LIN {X -0.179,Y -370.669,Z 1236.439,A 0.000,B 0.000,C 90.000,E1 79.106} C_DIS
LIN {X 0.099,Y -361.272,Z 1236.430,A 0.000,B 0.000,C 90.000,E1 77.297} C_DIS
LIN {X 0.011,Y -351.626,Z 1236.420,A 0.000,B 0.000,C 90.000,E1 75.519} C_DIS
LIN {X 0.097,Y -340.229,Z 1236.408,A 0.000,B 0.000,C 90.000,E1 73.378} C_DIS
LIN {X 0.001,Y -327.542,Z 1236.394,A 0.000,B 0.000,C 90.000,E1 70.913} C_DIS
LIN {X 0.007,Y -310.788,Z 1236.375,A 0.000,B 0.000,C 90.000,E1 67.411} C_DIS
LIN {X -0.044,Y -295.583,Z 1236.354,A 0.000,B 0.000,C 90.000,E1 63.819} C_DIS
LIN {X -0.046,Y -282.943,Z 1236.336,A 0.000,B 0.000,C 90.000,E1 60.461} C_DIS
LIN {X -0.122,Y -271.304,Z 1236.317,A 0.000,B 0.000,C 90.000,E1 57.041} C_DIS
LIN {X 0.053,Y -260.652,Z 1236.297,A 0.000,B 0.000,C 90.000,E1 53.497} C_DIS
LIN {X 0.109,Y -250.938,Z 1236.277,A 0.000,B 0.000,C 90.000,E1 49.908} C_DIS
LIN {X -0.029,Y -241.950,Z 1236.257,A 0.000,B 0.000,C 90.000,E1 46.296} C_DIS
LIN {X -0.042,Y -235.054,Z 1236.241,A 0.000,B 0.000,C 90.000,E1 43.338} C_DIS
LIN {X -0.040,Y -228.349,Z 1236.224,A 0.000,B 0.000,C 90.000,E1 40.334} C_DIS
LIN {X 0.029,Y -220.435,Z 1236.203,A 0.000,B 0.000,C 90.000,E1 36.503} C_DIS
LIN {X 0.039,Y -213.341,Z 1236.181,A 0.000,B 0.000,C 90.000,E1 32.625} C_DIS
LIN {X 0.035,Y -207.183,Z 1236.159,A 0.000,B 0.000,C 90.000,E1 28.693} C_DIS
LIN {X -0.003,Y -201.815,Z 1236.137,A 0.000,B 0.000,C 90.000,E1 24.719} C_DIS
LIN {X 0.088,Y -197.451,Z 1236.115,A 0.000,B 0.000,C 90.000,E1 20.663} C_DIS
LIN {X 0.056,Y -193.292,Z 1236.088,A 0.000,B 0.000,C 90.000,E1 15.788} C_DIS
LIN {X -0.068,Y -190.051,Z 1236.056,A 0.000,B 0.000,C 90.000,E1 10.074} C_DIS
LIN {X -0.056,Y -190.199,Z 1235.974,A 0.000,B 0.000,C 90.000,E1 355.412} C_DIS
LIN {X -0.017,Y -193.411,Z 1235.942,A 0.000,B 0.000,C 90.000,E1 349.634} C_DIS
LIN {X -0.111,Y -197.411,Z 1235.915,A 0.000,B 0.000,C 90.000,E1 344.755} C_DIS
LIN {X -0.029,Y -201.638,Z 1235.893,A 0.000,B 0.000,C 90.000,E1 340.678} C_DIS
LIN {X -0.040,Y -206.594,Z 1235.870,A 0.000,B 0.000,C 90.000,E1 336.666} C_DIS
LIN {X 0.069,Y -212.254,Z 1235.848,A 0.000,B 0.000,C 90.000,E1 332.666} C_DIS
LIN {X 0.023,Y -217.130,Z 1235.831,A 0.000,B 0.000,C 90.000,E1 329.537} C_DIS
LIN {X -0.042,Y -223.851,Z 1235.809,A 0.000,B 0.000,C 90.000,E1 325.674} C_DIS
LIN {X 0.063,Y -231.206,Z 1235.788,A 0.000,B 0.000,C 90.000,E1 321.823} C_DIS
LIN {X -0.030,Y -239.421,Z 1235.767,A 0.000,B 0.000,C 90.000,E1 318.081} C_DIS
LIN {X -0.074,Y -247.766,Z 1235.749,A 0.000,B 0.000,C 90.000,E1 314.757} C_DIS
LIN {X -0.018,Y -257.363,Z 1235.730,A 0.000,B 0.000,C 90.000,E1 311.472} C_DIS
LIN {X 0.156,Y -263.424,Z 1235.720,A 0.000,B 0.000,C 90.000,E1 309.644} C_DIS
LIN {X -0.140,Y -273.079,Z 1235.707,A 0.000,B 0.000,C 90.000,E1 307.237} C_DIS
LIN {X -0.057,Y -285.485,Z 1235.691,A 0.000,B 0.000,C 90.000,E1 304.452} C_DIS
LIN {X -0.050,Y -295.886,Z 1235.680,A 0.000,B 0.000,C 90.000,E1 302.418} C_DIS
LIN {X -0.011,Y -305.286,Z 1235.671,A 0.000,B 0.000,C 90.000,E1 300.747} C_DIS
LIN {X 0.082,Y -311.517,Z 1235.665,A 0.000,B 0.000,C 90.000,E1 299.745} C_DIS
LIN {X -0.191,Y -318.308,Z 1235.660,A 0.000,B 0.000,C 90.000,E1 298.821} C_DIS
LIN {X -0.131,Y -340.816,Z 1235.644,A 0.000,B 0.000,C 90.000,E1 295.976} C_DIS
LIN {X 0.057,Y -356.578,Z 1235.634,A 0.000,B 0.000,C 90.000,E1 294.131} C_DIS
LIN {X -0.042,Y -374.823,Z 1235.623,A 0.000,B 0.000,C 90.000,E1 292.153} C_DIS
LIN {X -0.141,Y -390.434,Z 1235.614,A 0.000,B 0.000,C 90.000,E1 290.482} C_DIS
LIN {X 0.066,Y -408.526,Z 1235.603,A 0.000,B 0.000,C 90.000,E1 288.544} C_DIS
LIN {X 0.208,Y -418.729,Z 1235.597,A 0.000,B 0.000,C 90.000,E1 287.457} C_DIS
LIN {X 0.098,Y -426.028,Z 1235.593,A 0.000,B 0.000,C 90.000,E1 286.677} C_DIS
LIN {X -0.103,Y -432.907,Z 1235.588,A 0.000,B 0.000,C 90.000,E1 285.898} C_DIS
LIN {X 0.145,Y -439.240,Z 1235.584,A 0.000,B 0.000,C 90.000,E1 285.064} C_DIS
LIN {X -0.092,Y -445.008,Z 1235.579,A 0.000,B 0.000,C 90.000,E1 284.300} C_DIS
LIN {X 0.164,Y -450.121,Z 1235.575,A 0.000,B 0.000,C 90.000,E1 283.480} C_DIS
LIN {X 0.027,Y -454.497,Z 1235.571,A 0.000,B 0.000,C 90.000,E1 282.715} C_DIS
LIN {X -0.069,Y -458.168,Z 1235.566,A 0.000,B 0.000,C 90.000,E1 281.951} C_DIS
LIN {X -0.139,Y -461.249,Z 1235.562,A 0.000,B 0.000,C 90.000,E1 281.186} C_DIS
LIN {X -0.027,Y -463.002,Z 1235.559,A 0.000,B 0.000,C 90.000,E1 280.658} C_DIS
LIN {X 0.014,Y -464.458,Z 1235.556,A 0.000,B 0.000,C 90.000,E1 280.141} C_DIS
LIN {X 0.148,Y -465.715,Z 1235.553,A 0.000,B 0.000,C 90.000,E1 279.613} C_DIS
LIN {X -0.247,Y -466.684,Z 1235.551,A 0.000,B 0.000,C 90.000,E1 279.151} C_DIS
LIN {X -0.102,Y -467.333,Z 1235.548,A 0.000,B 0.000,C 90.000,E1 278.624} C_DIS
LIN {X -0.024,Y -467.672,Z 1235.545,A 0.000,B 0.000,C 90.000,E1 278.106} C_DIS
LIN {X 0.062,Y -467.688,Z 1235.542,A 0.000,B 0.000,C 90.000,E1 277.587} C_DIS
LIN {X 0.152,Y -467.320,Z 1235.539,A 0.000,B 0.000,C 90.000,E1 277.068} C_DIS
LIN {X -0.222,Y -466.486,Z 1235.536,A 0.000,B 0.000,C 90.000,E1 276.606} C_DIS
LIN {X -0.133,Y -465.262,Z 1235.534,A 0.000,B 0.000,C 90.000,E1 276.087} C_DIS
LIN {X -0.051,Y -463.627,Z 1235.531,A 0.000,B 0.000,C 90.000,E1 275.568} C_DIS
LIN {X 0.023,Y -461.532,Z 1235.528,A 0.000,B 0.000,C 90.000,E1 275.049} C_DIS
LIN {X 0.086,Y -458.948,Z 1235.525,A 0.000,B 0.000,C 90.000,E1 274.531} C_DIS
LIN {X -0.139,Y -457.507,Z 1235.524,A 0.000,B 0.000,C 90.000,E1 274.302} C_DIS
LIN {X -0.105,Y -453.967,Z 1235.521,A 0.000,B 0.000,C 90.000,E1 273.784} C_DIS
LIN {X 0.119,Y -451.884,Z 1235.520,A 0.000,B 0.000,C 90.000,E1 273.498} C_DIS
LIN {X 0.119,Y -446.831,Z 1235.517,A 0.000,B 0.000,C 90.000,E1 272.980} C_DIS
LIN {X -0.189,Y -440.738,Z 1235.514,A 0.000,B 0.000,C 90.000,E1 272.522} C_DIS
LIN {X 0.061,Y -434.052,Z 1235.511,A 0.000,B 0.000,C 90.000,E1 272.064} C_DIS
LIN {X 0.003,Y -427.110,Z 1235.510,A 0.000,B 0.000,C 90.000,E1 271.718} C_DIS
LIN {X -0.030,Y -420.025,Z 1235.508,A 0.000,B 0.000,C 90.000,E1 271.432} C_DIS
LIN {X -0.120,Y -412.965,Z 1235.507,A 0.000,B 0.000,C 90.000,E1 271.203} C_DIS
LIN {X 0.061,Y -405.743,Z 1235.505,A 0.000,B 0.000,C 90.000,E1 270.974} C_DIS
LIN {X -0.013,Y -395.190,Z 1235.504,A 0.000,B 0.000,C 90.000,E1 270.745} C_DIS
LIN {X -0.148,Y -387.567,Z 1235.503,A 0.000,B 0.000,C 90.000,E1 270.630} C_DIS
LIN {X -0.120,Y -378.532,Z 1235.503,A 0.000,B 0.000,C 90.000,E1 270.516} C_DIS
LIN {X 0.140,Y -365.055,Z 1235.502,A 0.000,B 0.000,C 90.000,E1 270.401} C_DIS
LIN {X 0.082,Y -359.253,Z 1235.502,A 0.000,B 0.000,C 90.000,E1 270.401} C_DIS
LIN {X 0.013,Y -181.576,Z 1235.502,A 0.000,B 0.000,C 90.000,E1 270.401} C_DIS
LIN {X -0.055,Y -180.860,Z 1235.472,A 0.000,B 0.000,C 90.000,E1 265.008} C_DIS
LIN {X -0.001,Y -178.972,Z 1235.444,A 0.000,B 0.000,C 90.000,E1 259.926} C_DIS
LIN {X 0.008,Y -177.932,Z 1235.435,A 0.000,B 0.000,C 90.000,E1 258.229} C_DIS
LIN {X 0.024,Y -175.570,Z 1235.411,A 0.000,B 0.000,C 90.000,E1 253.976} C_DIS
LIN {X 0.030,Y -172.299,Z 1235.387,A 0.000,B 0.000,C 90.000,E1 249.699} C_DIS
LIN {X 0.008,Y -171.777,Z 1235.382,A 0.000,B 0.000,C 90.000,E1 248.847} C_DIS
LIN {X -0.020,Y -168.707,Z 1235.363,A 0.000,B 0.000,C 90.000,E1 245.409} C_DIS
LIN {X 0.019,Y -166.770,Z 1235.349,A 0.000,B 0.000,C 90.000,E1 242.794} C_DIS
LIN {X -0.061,Y -162.751,Z 1235.325,A 0.000,B 0.000,C 90.000,E1 238.456} C_DIS
LIN {X -0.085,Y -161.441,Z 1235.315,A 0.000,B 0.000,C 90.000,E1 236.707} C_DIS
LIN {X -0.042,Y -157.434,Z 1235.290,A 0.000,B 0.000,C 90.000,E1 232.271} C_DIS
LIN {X -0.009,Y -155.440,Z 1235.276,A 0.000,B 0.000,C 90.000,E1 229.585} C_DIS
LIN {X 0.040,Y -151.761,Z 1235.250,A 0.000,B 0.000,C 90.000,E1 225.081} C_DIS
LIN {X 0.052,Y -149.962,Z 1235.235,A 0.000,B 0.000,C 90.000,E1 222.366} C_DIS
LIN {X 0.079,Y -146.802,Z 1235.210,A 0.000,B 0.000,C 90.000,E1 217.810} C_DIS
LIN {X -0.021,Y -145.379,Z 1235.195,A 0.000,B 0.000,C 90.000,E1 215.105} C_DIS
LIN {X -0.029,Y -142.440,Z 1235.164,A 0.000,B 0.000,C 90.000,E1 209.589} C_DIS
LIN {X 0.018,Y -141.431,Z 1235.149,A 0.000,B 0.000,C 90.000,E1 206.796} C_DIS
LIN {X -0.001,Y -139.365,Z 1235.113,A 0.000,B 0.000,C 90.000,E1 200.301} C_DIS
LIN {X -0.015,Y -138.810,Z 1235.097,A 0.000,B 0.000,C 90.000,E1 197.511} C_DIS
LIN {X 0.037,Y -138.351,Z 1235.056,A 0.000,B 0.000,C 90.000,E1 190.018} C_DIS
LIN {X 0.012,Y -139.540,Z 1235.004,A 0.000,B 0.000,C 90.000,E1 180.688} C_DIS
LIN {X -0.035,Y -141.237,Z 1234.973,A 0.000,B 0.000,C 90.000,E1 175.122} C_DIS
LIN {X 0.065,Y -142.607,Z 1234.957,A 0.000,B 0.000,C 90.000,E1 172.299} C_DIS
LIN {X 0.018,Y -144.918,Z 1234.932,A 0.000,B 0.000,C 90.000,E1 167.701} C_DIS
LIN {X 0.010,Y -147.547,Z 1234.911,A 0.000,B 0.000,C 90.000,E1 164.031} C_DIS
LIN {X 0.042,Y -150.149,Z 1234.891,A 0.000,B 0.000,C 90.000,E1 160.369} C_DIS
LIN {X 0.052,Y -153.518,Z 1234.871,A 0.000,B 0.000,C 90.000,E1 156.741} C_DIS
LIN {X -0.027,Y -157.883,Z 1234.846,A 0.000,B 0.000,C 90.000,E1 152.281} C_DIS
LIN {X -0.073,Y -162.170,Z 1234.826,A 0.000,B 0.000,C 90.000,E1 148.742} C_DIS
LIN {X 0.042,Y -166.379,Z 1234.807,A 0.000,B 0.000,C 90.000,E1 145.182} C_DIS
LIN {X 0.044,Y -171.395,Z 1234.787,A 0.000,B 0.000,C 90.000,E1 141.698} C_DIS
LIN {X 0.084,Y -176.308,Z 1234.768,A 0.000,B 0.000,C 90.000,E1 138.243} C_DIS
LIN {X -0.047,Y -180.595,Z 1234.754,A 0.000,B 0.000,C 90.000,E1 135.729} C_DIS
LIN {X -0.070,Y -185.996,Z 1234.735,A 0.000,B 0.000,C 90.000,E1 132.366} C_DIS
LIN {X -0.015,Y -190.631,Z 1234.721,A 0.000,B 0.000,C 90.000,E1 129.850} C_DIS
LIN {X -0.108,Y -196.381,Z 1234.703,A 0.000,B 0.000,C 90.000,E1 126.583} C_DIS
LIN {X -0.039,Y -200.820,Z 1234.691,A 0.000,B 0.000,C 90.000,E1 124.326} C_DIS
LIN {X -0.097,Y -310.659,Z 1234.691,A 0.000,B 0.000,C 90.000,E1 124.326} C_DIS
LIN {X 0.055,Y -312.011,Z 1234.691,A 0.000,B 0.000,C 90.000,E1 124.278} C_DIS
LIN {X -0.050,Y -316.365,Z 1234.689,A 0.000,B 0.000,C 90.000,E1 124.119} C_DIS
LIN {X -0.061,Y -319.557,Z 1234.688,A 0.000,B 0.000,C 90.000,E1 123.865} C_DIS
LIN {X 0.074,Y -323.236,Z 1234.685,A 0.000,B 0.000,C 90.000,E1 123.372} C_DIS
LIN {X -0.116,Y -324.988,Z 1234.684,A 0.000,B 0.000,C 90.000,E1 123.086} C_DIS
LIN {X 0.064,Y -327.483,Z 1234.680,A 0.000,B 0.000,C 90.000,E1 122.418} C_DIS
LIN {X -0.062,Y -338.295,Z 1234.664,A 0.000,B 0.000,C 90.000,E1 119.617} C_DIS
LIN {X 0.094,Y -350.477,Z 1234.649,A 0.000,B 0.000,C 90.000,E1 116.821} C_DIS
LIN {X -0.046,Y -364.141,Z 1234.634,A 0.000,B 0.000,C 90.000,E1 114.131} C_DIS
LIN {X -0.036,Y -377.623,Z 1234.621,A 0.000,B 0.000,C 90.000,E1 111.770} C_DIS
LIN {X 0.042,Y -392.462,Z 1234.608,A 0.000,B 0.000,C 90.000,E1 109.450} C_DIS
LIN {X -0.139,Y -408.763,Z 1234.596,A 0.000,B 0.000,C 90.000,E1 107.221} C_DIS
LIN {X -0.043,Y -426.640,Z 1234.583,A 0.000,B 0.000,C 90.000,E1 105.009} C_DIS
LIN {X -0.058,Y -446.107,Z 1234.572,A 0.000,B 0.000,C 90.000,E1 102.883} C_DIS
LIN {X 0.091,Y -466.338,Z 1234.561,A 0.000,B 0.000,C 90.000,E1 100.894} C_DIS
LIN {X 0.104,Y -473.888,Z 1234.557,A 0.000,B 0.000,C 90.000,E1 100.197} C_DIS
LIN {X 0.163,Y -475.726,Z 1234.555,A 0.000,B 0.000,C 90.000,E1 99.962} C_DIS
LIN {X 0.028,Y -477.264,Z 1234.554,A 0.000,B 0.000,C 90.000,E1 99.726} C_DIS
LIN {X -0.188,Y -478.414,Z 1234.553,A 0.000,B 0.000,C 90.000,E1 99.500} C_DIS
LIN {X 0.029,Y -479.794,Z 1234.550,A 0.000,B 0.000,C 90.000,E1 98.973} C_DIS
LIN {X 0.179,Y -480.143,Z 1234.547,A 0.000,B 0.000,C 90.000,E1 98.454} C_DIS
LIN {X -0.136,Y -479.521,Z 1234.544,A 0.000,B 0.000,C 90.000,E1 97.992} C_DIS
LIN {X 0.028,Y -477.829,Z 1234.542,A 0.000,B 0.000,C 90.000,E1 97.473} C_DIS
LIN {X -0.099,Y -476.486,Z 1234.540,A 0.000,B 0.000,C 90.000,E1 97.239} C_DIS
LIN {X 0.205,Y -456.515,Z 1234.525,A 0.000,B 0.000,C 90.000,E1 94.416} C_DIS
LIN {X -0.017,Y -435.830,Z 1234.507,A 0.000,B 0.000,C 90.000,E1 91.318} C_DIS
LIN {X -0.015,Y -421.777,Z 1234.494,A 0.000,B 0.000,C 90.000,E1 88.912} C_DIS
LIN {X 0.142,Y -407.386,Z 1234.479,A 0.000,B 0.000,C 90.000,E1 86.159} C_DIS
LIN {X 0.166,Y -398.717,Z 1234.469,A 0.000,B 0.000,C 90.000,E1 84.489} C_DIS
LIN {X 0.046,Y -388.538,Z 1234.459,A 0.000,B 0.000,C 90.000,E1 82.534} C_DIS
LIN {X -0.155,Y -379.689,Z 1234.449,A 0.000,B 0.000,C 90.000,E1 80.849} C_DIS
LIN {X -0.131,Y -370.554,Z 1234.439,A 0.000,B 0.000,C 90.000,E1 79.106} C_DIS
LIN {X 0.144,Y -361.174,Z 1234.430,A 0.000,B 0.000,C 90.000,E1 77.297} C_DIS
LIN {X 0.054,Y -351.539,Z 1234.420,A 0.000,B 0.000,C 90.000,E1 75.519} C_DIS
LIN {X 0.131,Y -340.158,Z 1234.408,A 0.000,B 0.000,C 90.000,E1 73.378} C_DIS
LIN {X 0.032,Y -327.461,Z 1234.394,A 0.000,B 0.000,C 90.000,E1 70.913} C_DIS
LIN {X 0.039,Y -310.719,Z 1234.375,A 0.000,B 0.000,C 90.000,E1 67.411} C_DIS
LIN {X -0.021,Y -295.497,Z 1234.354,A 0.000,B 0.000,C 90.000,E1 63.819} C_DIS
LIN {X -0.025,Y -282.830,Z 1234.336,A 0.000,B 0.000,C 90.000,E1 60.461} C_DIS
LIN {X -0.106,Y -271.166,Z 1234.317,A 0.000,B 0.000,C 90.000,E1 57.041} C_DIS
LIN {X 0.011,Y -261.515,Z 1234.299,A 0.000,B 0.000,C 90.000,E1 53.863} C_DIS
LIN {X 0.092,Y -251.662,Z 1234.279,A 0.000,B 0.000,C 90.000,E1 50.275} C_DIS
LIN {X -0.019,Y -242.566,Z 1234.259,A 0.000,B 0.000,C 90.000,E1 46.662} C_DIS
LIN {X -0.018,Y -235.616,Z 1234.243,A 0.000,B 0.000,C 90.000,E1 43.704} C_DIS
LIN {X -0.007,Y -228.841,Z 1234.226,A 0.000,B 0.000,C 90.000,E1 40.701} C_DIS
LIN {X 0.076,Y -220.821,Z 1234.205,A 0.000,B 0.000,C 90.000,E1 36.870} C_DIS
LIN {X 0.037,Y -213.626,Z 1234.183,A 0.000,B 0.000,C 90.000,E1 33.007} C_DIS
LIN {X 0.035,Y -207.364,Z 1234.162,A 0.000,B 0.000,C 90.000,E1 29.077} C_DIS
LIN {X 0.086,Y -201.921,Z 1234.139,A 0.000,B 0.000,C 90.000,E1 25.079} C_DIS
LIN {X -0.084,Y -197.485,Z 1234.117,A 0.000,B 0.000,C 90.000,E1 21.099} C_DIS
LIN {X -0.049,Y -193.258,Z 1234.090,A 0.000,B 0.000,C 90.000,E1 16.205} C_DIS
LIN {X 0.021,Y -189.906,Z 1234.058,A 0.000,B 0.000,C 90.000,E1 10.433} C_DIS
LIN {X -0.066,Y -189.895,Z 1233.974,A 0.000,B 0.000,C 90.000,E1 355.412} C_DIS
LIN {X -0.040,Y -193.110,Z 1233.942,A 0.000,B 0.000,C 90.000,E1 349.634} C_DIS
LIN {X 0.045,Y -197.146,Z 1233.915,A 0.000,B 0.000,C 90.000,E1 344.700} C_DIS
LIN {X -0.072,Y -201.405,Z 1233.893,A 0.000,B 0.000,C 90.000,E1 340.678} C_DIS
LIN {X -0.092,Y -206.388,Z 1233.870,A 0.000,B 0.000,C 90.000,E1 336.666} C_DIS
LIN {X 0.010,Y -212.074,Z 1233.848,A 0.000,B 0.000,C 90.000,E1 332.666} C_DIS
LIN {X -0.042,Y -216.971,Z 1233.831,A 0.000,B 0.000,C 90.000,E1 329.537} C_DIS
LIN {X -0.115,Y -223.693,Z 1233.809,A 0.000,B 0.000,C 90.000,E1 325.674} C_DIS
LIN {X -0.016,Y -231.058,Z 1233.788,A 0.000,B 0.000,C 90.000,E1 321.823} C_DIS
LIN {X -0.117,Y -239.295,Z 1233.767,A 0.000,B 0.000,C 90.000,E1 318.081} C_DIS
LIN {X 0.007,Y -247.637,Z 1233.748,A 0.000,B 0.000,C 90.000,E1 314.717} C_DIS
LIN {X 0.052,Y -257.323,Z 1233.730,A 0.000,B 0.000,C 90.000,E1 311.434} C_DIS
LIN {X 0.052,Y -263.406,Z 1233.720,A 0.000,B 0.000,C 90.000,E1 309.644} C_DIS
LIN {X 0.059,Y -271.585,Z 1233.708,A 0.000,B 0.000,C 90.000,E1 307.523} C_DIS
LIN {X 0.112,Y -283.813,Z 1233.693,A 0.000,B 0.000,C 90.000,E1 304.739} C_DIS
LIN {X -0.153,Y -294.033,Z 1233.682,A 0.000,B 0.000,C 90.000,E1 302.752} C_DIS
LIN {X 0.045,Y -307.186,Z 1233.669,A 0.000,B 0.000,C 90.000,E1 300.384} C_DIS
LIN {X 0.051,Y -315.845,Z 1233.662,A 0.000,B 0.000,C 90.000,E1 299.077} C_DIS
LIN {X -0.089,Y -330.556,Z 1233.651,A 0.000,B 0.000,C 90.000,E1 297.180} C_DIS
LIN {X -0.023,Y -351.460,Z 1233.637,A 0.000,B 0.000,C 90.000,E1 294.695} C_DIS
LIN {X -0.082,Y -372.485,Z 1233.624,A 0.000,B 0.000,C 90.000,E1 292.386} C_DIS
LIN {X 0.044,Y -385.457,Z 1233.617,A 0.000,B 0.000,C 90.000,E1 290.972} C_DIS
LIN {X 0.068,Y -400.947,Z 1233.607,A 0.000,B 0.000,C 90.000,E1 289.322} C_DIS
LIN {X -0.102,Y -416.183,Z 1233.599,A 0.000,B 0.000,C 90.000,E1 287.764} C_DIS
LIN {X -0.170,Y -423.544,Z 1233.594,A 0.000,B 0.000,C 90.000,E1 286.985} C_DIS
LIN {X 0.126,Y -430.616,Z 1233.590,A 0.000,B 0.000,C 90.000,E1 286.134} C_DIS
LIN {X -0.190,Y -437.164,Z 1233.585,A 0.000,B 0.000,C 90.000,E1 285.371} C_DIS
LIN {X 0.100,Y -443.139,Z 1233.581,A 0.000,B 0.000,C 90.000,E1 284.537} C_DIS
LIN {X -0.102,Y -448.488,Z 1233.576,A 0.000,B 0.000,C 90.000,E1 283.772} C_DIS
LIN {X -0.252,Y -453.115,Z 1233.572,A 0.000,B 0.000,C 90.000,E1 283.008} C_DIS
LIN {X 0.081,Y -457.053,Z 1233.568,A 0.000,B 0.000,C 90.000,E1 282.187} C_DIS
LIN {X 0.177,Y -459.309,Z 1233.565,A 0.000,B 0.000,C 90.000,E1 281.658} C_DIS
LIN {X -0.166,Y -461.321,Z 1233.562,A 0.000,B 0.000,C 90.000,E1 281.186} C_DIS
LIN {X -0.053,Y -463.056,Z 1233.559,A 0.000,B 0.000,C 90.000,E1 280.658} C_DIS
LIN {X -0.012,Y -464.544,Z 1233.556,A 0.000,B 0.000,C 90.000,E1 280.141} C_DIS
LIN {X 0.122,Y -465.775,Z 1233.553,A 0.000,B 0.000,C 90.000,E1 279.613} C_DIS
LIN {X 0.187,Y -466.740,Z 1233.551,A 0.000,B 0.000,C 90.000,E1 279.095} C_DIS
LIN {X -0.128,Y -467.409,Z 1233.548,A 0.000,B 0.000,C 90.000,E1 278.624} C_DIS
LIN {X -0.048,Y -467.738,Z 1233.545,A 0.000,B 0.000,C 90.000,E1 278.106} C_DIS
LIN {X 0.038,Y -467.771,Z 1233.542,A 0.000,B 0.000,C 90.000,E1 277.587} C_DIS
LIN {X 0.127,Y -467.425,Z 1233.539,A 0.000,B 0.000,C 90.000,E1 277.068} C_DIS
LIN {X -0.246,Y -466.634,Z 1233.536,A 0.000,B 0.000,C 90.000,E1 276.606} C_DIS
LIN {X -0.157,Y -465.424,Z 1233.534,A 0.000,B 0.000,C 90.000,E1 276.087} C_DIS
LIN {X -0.073,Y -463.810,Z 1233.531,A 0.000,B 0.000,C 90.000,E1 275.568} C_DIS
LIN {X 0.002,Y -461.752,Z 1233.528,A 0.000,B 0.000,C 90.000,E1 275.049} C_DIS
LIN {X 0.066,Y -459.211,Z 1233.525,A 0.000,B 0.000,C 90.000,E1 274.531} C_DIS
LIN {X 0.108,Y -456.028,Z 1233.522,A 0.000,B 0.000,C 90.000,E1 274.012} C_DIS
LIN {X -0.122,Y -454.235,Z 1233.521,A 0.000,B 0.000,C 90.000,E1 273.784} C_DIS
LIN {X -0.134,Y -449.779,Z 1233.518,A 0.000,B 0.000,C 90.000,E1 273.269} C_DIS
LIN {X 0.104,Y -447.141,Z 1233.517,A 0.000,B 0.000,C 90.000,E1 272.980} C_DIS
LIN {X -0.052,Y -444.258,Z 1233.515,A 0.000,B 0.000,C 90.000,E1 272.751} C_DIS
LIN {X -0.206,Y -441.029,Z 1233.514,A 0.000,B 0.000,C 90.000,E1 272.522} C_DIS
LIN {X -0.073,Y -437.910,Z 1233.513,A 0.000,B 0.000,C 90.000,E1 272.293} C_DIS
LIN {X 0.043,Y -431.264,Z 1233.510,A 0.000,B 0.000,C 90.000,E1 271.892} C_DIS
LIN {X -0.187,Y -424.334,Z 1233.509,A 0.000,B 0.000,C 90.000,E1 271.604} C_DIS
LIN {X -0.038,Y -417.274,Z 1233.507,A 0.000,B 0.000,C 90.000,E1 271.318} C_DIS
LIN {X -0.001,Y -410.222,Z 1233.506,A 0.000,B 0.000,C 90.000,E1 271.088} C_DIS
LIN {X 0.090,Y -399.224,Z 1233.505,A 0.000,B 0.000,C 90.000,E1 270.802} C_DIS
LIN {X -0.119,Y -392.469,Z 1233.504,A 0.000,B 0.000,C 90.000,E1 270.688} C_DIS
LIN {X 0.146,Y -383.655,Z 1233.503,A 0.000,B 0.000,C 90.000,E1 270.516} C_DIS
LIN {X 0.141,Y -370.172,Z 1233.502,A 0.000,B 0.000,C 90.000,E1 270.401} C_DIS
LIN {X 0.024,Y -364.814,Z 1233.502,A 0.000,B 0.000,C 90.000,E1 270.401} C_DIS
LIN {X -0.017,Y -181.576,Z 1233.502,A 0.000,B 0.000,C 90.000,E1 270.401} C_DIS
LIN {X -0.087,Y -180.858,Z 1233.472,A 0.000,B 0.000,C 90.000,E1 265.008} C_DIS
LIN {X -0.033,Y -178.969,Z 1233.444,A 0.000,B 0.000,C 90.000,E1 259.926} C_DIS
LIN {X -0.023,Y -177.925,Z 1233.435,A 0.000,B 0.000,C 90.000,E1 258.229} C_DIS
LIN {X -0.008,Y -175.562,Z 1233.411,A 0.000,B 0.000,C 90.000,E1 253.976} C_DIS
LIN {X 0.000,Y -172.292,Z 1233.387,A 0.000,B 0.000,C 90.000,E1 249.699} C_DIS
LIN {X -0.022,Y -171.771,Z 1233.382,A 0.000,B 0.000,C 90.000,E1 248.847} C_DIS
LIN {X -0.031,Y -168.012,Z 1233.359,A 0.000,B 0.000,C 90.000,E1 244.537} C_DIS
LIN {X -0.011,Y -166.762,Z 1233.349,A 0.000,B 0.000,C 90.000,E1 242.794} C_DIS
LIN {X 0.048,Y -162.742,Z 1233.325,A 0.000,B 0.000,C 90.000,E1 238.408} C_DIS
LIN {X 0.109,Y -161.433,Z 1233.315,A 0.000,B 0.000,C 90.000,E1 236.628} C_DIS
LIN {X -0.071,Y -157.426,Z 1233.290,A 0.000,B 0.000,C 90.000,E1 232.271} C_DIS
LIN {X -0.037,Y -155.430,Z 1233.275,A 0.000,B 0.000,C 90.000,E1 229.585} C_DIS
LIN {X 0.012,Y -151.753,Z 1233.250,A 0.000,B 0.000,C 90.000,E1 225.081} C_DIS
LIN {X 0.023,Y -149.954,Z 1233.235,A 0.000,B 0.000,C 90.000,E1 222.366} C_DIS
LIN {X 0.050,Y -146.797,Z 1233.210,A 0.000,B 0.000,C 90.000,E1 217.810} C_DIS
LIN {X -0.049,Y -145.371,Z 1233.195,A 0.000,B 0.000,C 90.000,E1 215.105} C_DIS
LIN {X 0.068,Y -142.435,Z 1233.164,A 0.000,B 0.000,C 90.000,E1 209.539} C_DIS
LIN {X -0.010,Y -141.425,Z 1233.149,A 0.000,B 0.000,C 90.000,E1 206.796} C_DIS
LIN {X -0.028,Y -139.363,Z 1233.113,A 0.000,B 0.000,C 90.000,E1 200.301} C_DIS
LIN {X -0.041,Y -138.808,Z 1233.097,A 0.000,B 0.000,C 90.000,E1 197.511} C_DIS
LIN {X 0.009,Y -138.350,Z 1233.056,A 0.000,B 0.000,C 90.000,E1 190.018} C_DIS
LIN {X -0.015,Y -139.543,Z 1233.004,A 0.000,B 0.000,C 90.000,E1 180.688} C_DIS
LIN {X -0.062,Y -141.241,Z 1232.973,A 0.000,B 0.000,C 90.000,E1 175.122} C_DIS
LIN {X 0.037,Y -142.611,Z 1232.957,A 0.000,B 0.000,C 90.000,E1 172.299} C_DIS
LIN {X -0.011,Y -144.924,Z 1232.932,A 0.000,B 0.000,C 90.000,E1 167.701} C_DIS
LIN {X -0.018,Y -147.553,Z 1232.911,A 0.000,B 0.000,C 90.000,E1 164.031} C_DIS
LIN {X 0.014,Y -150.158,Z 1232.891,A 0.000,B 0.000,C 90.000,E1 160.369} C_DIS
LIN {X 0.023,Y -153.529,Z 1232.871,A 0.000,B 0.000,C 90.000,E1 156.741} C_DIS
LIN {X 0.075,Y -156.947,Z 1232.851,A 0.000,B 0.000,C 90.000,E1 153.127} C_DIS
LIN {X 0.012,Y -161.051,Z 1232.831,A 0.000,B 0.000,C 90.000,E1 149.587} C_DIS
LIN {X 0.097,Y -163.161,Z 1232.821,A 0.000,B 0.000,C 90.000,E1 147.788} C_DIS
LIN {X -0.032,Y -167.578,Z 1232.802,A 0.000,B 0.000,C 90.000,E1 144.322} C_DIS
LIN {X 0.014,Y -171.408,Z 1232.787,A 0.000,B 0.000,C 90.000,E1 141.698} C_DIS
LIN {X 0.053,Y -176.324,Z 1232.768,A 0.000,B 0.000,C 90.000,E1 138.243} C_DIS
LIN {X -0.079,Y -180.612,Z 1232.754,A 0.000,B 0.000,C 90.000,E1 135.729} C_DIS
LIN {X 0.036,Y -186.013,Z 1232.735,A 0.000,B 0.000,C 90.000,E1 132.324} C_DIS
LIN {X -0.048,Y -190.648,Z 1232.721,A 0.000,B 0.000,C 90.000,E1 129.850} C_DIS
LIN {X 0.016,Y -196.399,Z 1232.703,A 0.000,B 0.000,C 90.000,E1 126.537} C_DIS
LIN {X 0.045,Y -200.862,Z 1232.691,A 0.000,B 0.000,C 90.000,E1 124.278} C_DIS
LIN {X 0.035,Y -310.473,Z 1232.690,A 0.000,B 0.000,C 90.000,E1 124.278} C_DIS
LIN {X -0.103,Y -316.182,Z 1232.689,A 0.000,B 0.000,C 90.000,E1 124.119} C_DIS
LIN {X 0.067,Y -319.128,Z 1232.688,A 0.000,B 0.000,C 90.000,E1 123.865} C_DIS
LIN {X 0.054,Y -322.861,Z 1232.686,A 0.000,B 0.000,C 90.000,E1 123.420} C_DIS
LIN {X 0.142,Y -324.707,Z 1232.684,A 0.000,B 0.000,C 90.000,E1 123.086} C_DIS
LIN {X -0.043,Y -326.141,Z 1232.682,A 0.000,B 0.000,C 90.000,E1 122.801} C_DIS
LIN {X -0.087,Y -338.087,Z 1232.665,A 0.000,B 0.000,C 90.000,E1 119.667} C_DIS
LIN {X 0.054,Y -350.244,Z 1232.649,A 0.000,B 0.000,C 90.000,E1 116.873} C_DIS
LIN {X 0.082,Y -363.882,Z 1232.634,A 0.000,B 0.000,C 90.000,E1 114.155} C_DIS
LIN {X 0.105,Y -377.341,Z 1232.621,A 0.000,B 0.000,C 90.000,E1 111.791} C_DIS
LIN {X -0.043,Y -392.154,Z 1232.608,A 0.000,B 0.000,C 90.000,E1 109.504} C_DIS
LIN {X 0.149,Y -408.427,Z 1232.596,A 0.000,B 0.000,C 90.000,E1 107.221} C_DIS
LIN {X -0.162,Y -426.275,Z 1232.584,A 0.000,B 0.000,C 90.000,E1 105.064} C_DIS
LIN {X 0.230,Y -445.719,Z 1232.572,A 0.000,B 0.000,C 90.000,E1 102.883} C_DIS
LIN {X -0.092,Y -465.940,Z 1232.561,A 0.000,B 0.000,C 90.000,E1 100.950} C_DIS
LIN {X -0.091,Y -473.536,Z 1232.557,A 0.000,B 0.000,C 90.000,E1 100.254} C_DIS
LIN {X -0.036,Y -475.432,Z 1232.556,A 0.000,B 0.000,C 90.000,E1 100.018} C_DIS
LIN {X -0.174,Y -477.014,Z 1232.554,A 0.000,B 0.000,C 90.000,E1 99.782} C_DIS
LIN {X 0.080,Y -478.199,Z 1232.553,A 0.000,B 0.000,C 90.000,E1 99.500} C_DIS
LIN {X -0.176,Y -479.633,Z 1232.550,A 0.000,B 0.000,C 90.000,E1 99.029} C_DIS
LIN {X -0.029,Y -480.029,Z 1232.547,A 0.000,B 0.000,C 90.000,E1 98.511} C_DIS
LIN {X 0.130,Y -479.455,Z 1232.544,A 0.000,B 0.000,C 90.000,E1 97.992} C_DIS
LIN {X -0.183,Y -477.821,Z 1232.542,A 0.000,B 0.000,C 90.000,E1 97.530} C_DIS
LIN {X 0.164,Y -476.516,Z 1232.540,A 0.000,B 0.000,C 90.000,E1 97.239} C_DIS
LIN {X -0.028,Y -469.151,Z 1232.535,A 0.000,B 0.000,C 90.000,E1 96.258} C_DIS
LIN {X -0.204,Y -451.285,Z 1232.521,A 0.000,B 0.000,C 90.000,E1 93.726} C_DIS
LIN {X 0.113,Y -432.606,Z 1232.505,A 0.000,B 0.000,C 90.000,E1 90.802} C_DIS
LIN {X 0.031,Y -418.836,Z 1232.491,A 0.000,B 0.000,C 90.000,E1 88.396} C_DIS
LIN {X 0.063,Y -405.957,Z 1232.477,A 0.000,B 0.000,C 90.000,E1 85.927} C_DIS
LIN {X 0.101,Y -395.815,Z 1232.467,A 0.000,B 0.000,C 90.000,E1 83.970} C_DIS
LIN {X -0.027,Y -385.623,Z 1232.456,A 0.000,B 0.000,C 90.000,E1 82.008} C_DIS
LIN {X 0.041,Y -376.690,Z 1232.446,A 0.000,B 0.000,C 90.000,E1 80.274} C_DIS
LIN {X 0.069,Y -367.466,Z 1232.436,A 0.000,B 0.000,C 90.000,E1 78.522} C_DIS
LIN {X -0.036,Y -359.628,Z 1232.428,A 0.000,B 0.000,C 90.000,E1 77.061} C_DIS
LIN {X -0.149,Y -349.963,Z 1232.418,A 0.000,B 0.000,C 90.000,E1 75.283} C_DIS
LIN {X -0.099,Y -337.033,Z 1232.405,A 0.000,B 0.000,C 90.000,E1 72.834} C_DIS
LIN {X 0.041,Y -324.360,Z 1232.391,A 0.000,B 0.000,C 90.000,E1 70.315} C_DIS
LIN {X 0.054,Y -307.893,Z 1232.371,A 0.000,B 0.000,C 90.000,E1 66.794} C_DIS
LIN {X 0.026,Y -292.887,Z 1232.351,A 0.000,B 0.000,C 90.000,E1 63.179} C_DIS
LIN {X 0.075,Y -280.397,Z 1232.332,A 0.000,B 0.000,C 90.000,E1 59.793} C_DIS
LIN {X 0.065,Y -268.931,Z 1232.313,A 0.000,B 0.000,C 90.000,E1 56.342} C_DIS
LIN {X -0.096,Y -259.380,Z 1232.296,A 0.000,B 0.000,C 90.000,E1 53.210} C_DIS
LIN {X -0.076,Y -249.640,Z 1232.276,A 0.000,B 0.000,C 90.000,E1 49.622} C_DIS
LIN {X -0.087,Y -240.611,Z 1232.255,A 0.000,B 0.000,C 90.000,E1 45.972} C_DIS
LIN {X 0.028,Y -233.635,Z 1232.239,A 0.000,B 0.000,C 90.000,E1 42.975} C_DIS
LIN {X 0.009,Y -226.893,Z 1232.222,A 0.000,B 0.000,C 90.000,E1 39.967} C_DIS
LIN {X 0.031,Y -218.996,Z 1232.201,A 0.000,B 0.000,C 90.000,E1 36.137} C_DIS
LIN {X -0.010,Y -211.970,Z 1232.179,A 0.000,B 0.000,C 90.000,E1 32.260} C_DIS
LIN {X 0.016,Y -205.849,Z 1232.157,A 0.000,B 0.000,C 90.000,E1 28.309} C_DIS
LIN {X -0.060,Y -200.622,Z 1232.135,A 0.000,B 0.000,C 90.000,E1 24.335} C_DIS
LIN {X -0.080,Y -196.389,Z 1232.113,A 0.000,B 0.000,C 90.000,E1 20.301} C_DIS
LIN {X 0.038,Y -192.365,Z 1232.085,A 0.000,B 0.000,C 90.000,E1 15.371} C_DIS
LIN {X 0.024,Y -189.273,Z 1232.053,A 0.000,B 0.000,C 90.000,E1 9.613} C_DIS
LIN {X -0.020,Y -190.334,Z 1231.965,A 0.000,B 0.000,C 90.000,E1 353.742} C_DIS
LIN {X -0.068,Y -193.418,Z 1231.938,A 0.000,B 0.000,C 90.000,E1 348.814} C_DIS
LIN {X 0.078,Y -197.653,Z 1231.911,A 0.000,B 0.000,C 90.000,E1 343.866} C_DIS
LIN {X 0.013,Y -203.055,Z 1231.884,A 0.000,B 0.000,C 90.000,E1 339.028} C_DIS
LIN {X -0.066,Y -208.379,Z 1231.861,A 0.000,B 0.000,C 90.000,E1 335.049} C_DIS
LIN {X 0.094,Y -214.332,Z 1231.839,A 0.000,B 0.000,C 90.000,E1 331.051} C_DIS
LIN {X 0.016,Y -220.743,Z 1231.818,A 0.000,B 0.000,C 90.000,E1 327.168} C_DIS
LIN {X 0.075,Y -226.418,Z 1231.801,A 0.000,B 0.000,C 90.000,E1 324.069} C_DIS
LIN {X 0.039,Y -234.116,Z 1231.779,A 0.000,B 0.000,C 90.000,E1 320.275} C_DIS
LIN {X 0.012,Y -242.726,Z 1231.759,A 0.000,B 0.000,C 90.000,E1 316.539} C_DIS
LIN {X 0.070,Y -249.570,Z 1231.744,A 0.000,B 0.000,C 90.000,E1 313.947} C_DIS
LIN {X -0.019,Y -258.415,Z 1231.728,A 0.000,B 0.000,C 90.000,E1 311.067} C_DIS
LIN {X 0.113,Y -267.376,Z 1231.714,A 0.000,B 0.000,C 90.000,E1 308.543} C_DIS
LIN {X 0.110,Y -274.506,Z 1231.704,A 0.000,B 0.000,C 90.000,E1 306.790} C_DIS
LIN {X -0.051,Y -285.455,Z 1231.691,A 0.000,B 0.000,C 90.000,E1 304.405} C_DIS
LIN {X 0.119,Y -295.839,Z 1231.680,A 0.000,B 0.000,C 90.000,E1 302.339} C_DIS
LIN {X -0.082,Y -307.097,Z 1231.669,A 0.000,B 0.000,C 90.000,E1 300.384} C_DIS
LIN {X -0.080,Y -315.727,Z 1231.661,A 0.000,B 0.000,C 90.000,E1 299.077} C_DIS
LIN {X 0.029,Y -327.869,Z 1231.653,A 0.000,B 0.000,C 90.000,E1 297.462} C_DIS
LIN {X 0.120,Y -348.768,Z 1231.639,A 0.000,B 0.000,C 90.000,E1 294.951} C_DIS
LIN {X -0.103,Y -369.876,Z 1231.626,A 0.000,B 0.000,C 90.000,E1 292.642} C_DIS
LIN {X 0.017,Y -382.967,Z 1231.618,A 0.000,B 0.000,C 90.000,E1 291.227} C_DIS
LIN {X -0.054,Y -398.559,Z 1231.609,A 0.000,B 0.000,C 90.000,E1 289.577} C_DIS
LIN {X -0.134,Y -413.956,Z 1231.600,A 0.000,B 0.000,C 90.000,E1 288.000} C_DIS
LIN {X 0.208,Y -423.652,Z 1231.594,A 0.000,B 0.000,C 90.000,E1 286.913} C_DIS
LIN {X -0.026,Y -430.735,Z 1231.590,A 0.000,B 0.000,C 90.000,E1 286.134} C_DIS
LIN {X 0.079,Y -437.282,Z 1231.585,A 0.000,B 0.000,C 90.000,E1 285.315} C_DIS
LIN {X -0.055,Y -443.252,Z 1231.581,A 0.000,B 0.000,C 90.000,E1 284.537} C_DIS
LIN {X -0.257,Y -448.583,Z 1231.576,A 0.000,B 0.000,C 90.000,E1 283.772} C_DIS
LIN {X 0.136,Y -453.227,Z 1231.572,A 0.000,B 0.000,C 90.000,E1 282.939} C_DIS
LIN {X -0.075,Y -457.175,Z 1231.568,A 0.000,B 0.000,C 90.000,E1 282.187} C_DIS
LIN {X 0.021,Y -459.457,Z 1231.565,A 0.000,B 0.000,C 90.000,E1 281.658} C_DIS
LIN {X 0.131,Y -461.452,Z 1231.562,A 0.000,B 0.000,C 90.000,E1 281.130} C_DIS
LIN {X -0.208,Y -463.183,Z 1231.559,A 0.000,B 0.000,C 90.000,E1 280.658} C_DIS
LIN {X -0.167,Y -464.665,Z 1231.556,A 0.000,B 0.000,C 90.000,E1 280.141} C_DIS
LIN {X -0.032,Y -465.894,Z 1231.553,A 0.000,B 0.000,C 90.000,E1 279.613} C_DIS
LIN {X 0.033,Y -466.855,Z 1231.551,A 0.000,B 0.000,C 90.000,E1 279.095} C_DIS
LIN {X 0.180,Y -467.482,Z 1231.548,A 0.000,B 0.000,C 90.000,E1 278.568} C_DIS
LIN {X -0.202,Y -467.860,Z 1231.545,A 0.000,B 0.000,C 90.000,E1 278.106} C_DIS
LIN {X -0.115,Y -467.884,Z 1231.542,A 0.000,B 0.000,C 90.000,E1 277.587} C_DIS
LIN {X -0.025,Y -467.509,Z 1231.539,A 0.000,B 0.000,C 90.000,E1 277.068} C_DIS
LIN {X 0.067,Y -466.748,Z 1231.536,A 0.000,B 0.000,C 90.000,E1 276.549} C_DIS
LIN {X 0.156,Y -465.563,Z 1231.534,A 0.000,B 0.000,C 90.000,E1 276.030} C_DIS
LIN {X -0.223,Y -463.927,Z 1231.531,A 0.000,B 0.000,C 90.000,E1 275.568} C_DIS
LIN {X -0.146,Y -461.899,Z 1231.528,A 0.000,B 0.000,C 90.000,E1 275.049} C_DIS
LIN {X -0.081,Y -459.316,Z 1231.525,A 0.000,B 0.000,C 90.000,E1 274.531} C_DIS
LIN {X 0.153,Y -457.903,Z 1231.524,A 0.000,B 0.000,C 90.000,E1 274.245} C_DIS
LIN {X 0.187,Y -454.384,Z 1231.521,A 0.000,B 0.000,C 90.000,E1 273.726} C_DIS
LIN {X 0.174,Y -449.912,Z 1231.518,A 0.000,B 0.000,C 90.000,E1 273.212} C_DIS
LIN {X -0.173,Y -444.395,Z 1231.515,A 0.000,B 0.000,C 90.000,E1 272.751} C_DIS
LIN {X -0.153,Y -438.139,Z 1231.513,A 0.000,B 0.000,C 90.000,E1 272.293} C_DIS
LIN {X -0.017,Y -431.480,Z 1231.510,A 0.000,B 0.000,C 90.000,E1 271.892} C_DIS
LIN {X 0.178,Y -424.525,Z 1231.509,A 0.000,B 0.000,C 90.000,E1 271.547} C_DIS
LIN {X -0.095,Y -417.496,Z 1231.507,A 0.000,B 0.000,C 90.000,E1 271.318} C_DIS
LIN {X -0.066,Y -410.373,Z 1231.506,A 0.000,B 0.000,C 90.000,E1 271.088} C_DIS
LIN {X -0.008,Y -399.267,Z 1231.504,A 0.000,B 0.000,C 90.000,E1 270.802} C_DIS
LIN {X 0.169,Y -392.483,Z 1231.504,A 0.000,B 0.000,C 90.000,E1 270.630} C_DIS
LIN {X 0.058,Y -383.947,Z 1231.503,A 0.000,B 0.000,C 90.000,E1 270.516} C_DIS
LIN {X 0.053,Y -370.851,Z 1231.502,A 0.000,B 0.000,C 90.000,E1 270.401} C_DIS
LIN {X -0.122,Y -362.366,Z 1231.502,A 0.000,B 0.000,C 90.000,E1 270.401} C_DIS
LIN {X -0.090,Y -181.578,Z 1231.502,A 0.000,B 0.000,C 90.000,E1 270.401} C_DIS
LIN {X 0.047,Y -180.854,Z 1231.472,A 0.000,B 0.000,C 90.000,E1 264.951} C_DIS
LIN {X -0.079,Y -178.965,Z 1231.444,A 0.000,B 0.000,C 90.000,E1 259.926} C_DIS
LIN {X -0.068,Y -177.915,Z 1231.434,A 0.000,B 0.000,C 90.000,E1 258.229} C_DIS
LIN {X -0.053,Y -175.551,Z 1231.411,A 0.000,B 0.000,C 90.000,E1 253.976} C_DIS
LIN {X -0.045,Y -172.283,Z 1231.387,A 0.000,B 0.000,C 90.000,E1 249.699} C_DIS
LIN {X -0.006,Y -171.761,Z 1231.382,A 0.000,B 0.000,C 90.000,E1 248.827} C_DIS
LIN {X 0.011,Y -167.361,Z 1231.354,A 0.000,B 0.000,C 90.000,E1 243.640} C_DIS
LIN {X -0.055,Y -166.751,Z 1231.349,A 0.000,B 0.000,C 90.000,E1 242.794} C_DIS
LIN {X 0.005,Y -162.730,Z 1231.324,A 0.000,B 0.000,C 90.000,E1 238.408} C_DIS
LIN {X 0.066,Y -161.420,Z 1231.315,A 0.000,B 0.000,C 90.000,E1 236.628} C_DIS
LIN {X 0.107,Y -157.413,Z 1231.290,A 0.000,B 0.000,C 90.000,E1 232.190} C_DIS
LIN {X 0.040,Y -155.415,Z 1231.275,A 0.000,B 0.000,C 90.000,E1 229.542} C_DIS
LIN {X -0.029,Y -151.742,Z 1231.250,A 0.000,B 0.000,C 90.000,E1 225.081} C_DIS
LIN {X -0.018,Y -149.941,Z 1231.235,A 0.000,B 0.000,C 90.000,E1 222.366} C_DIS
LIN {X 0.011,Y -146.787,Z 1231.210,A 0.000,B 0.000,C 90.000,E1 217.810} C_DIS
LIN {X -0.089,Y -145.361,Z 1231.195,A 0.000,B 0.000,C 90.000,E1 215.105} C_DIS
LIN {X 0.027,Y -142.429,Z 1231.164,A 0.000,B 0.000,C 90.000,E1 209.539} C_DIS
LIN {X 0.078,Y -141.417,Z 1231.149,A 0.000,B 0.000,C 90.000,E1 206.744} C_DIS
LIN {X -0.067,Y -139.361,Z 1231.113,A 0.000,B 0.000,C 90.000,E1 200.301} C_DIS
LIN {X 0.052,Y -138.804,Z 1231.097,A 0.000,B 0.000,C 90.000,E1 197.457} C_DIS
LIN {X -0.030,Y -138.349,Z 1231.056,A 0.000,B 0.000,C 90.000,E1 190.018} C_DIS
LIN {X -0.054,Y -139.545,Z 1231.004,A 0.000,B 0.000,C 90.000,E1 180.688} C_DIS
LIN {X 0.038,Y -141.248,Z 1230.973,A 0.000,B 0.000,C 90.000,E1 175.065} C_DIS
LIN {X -0.003,Y -142.618,Z 1230.957,A 0.000,B 0.000,C 90.000,E1 172.299} C_DIS
LIN {X -0.050,Y -144.935,Z 1230.932,A 0.000,B 0.000,C 90.000,E1 167.701} C_DIS
LIN {X 0.083,Y -147.564,Z 1230.911,A 0.000,B 0.000,C 90.000,E1 163.976} C_DIS
LIN {X -0.028,Y -150.171,Z 1230.891,A 0.000,B 0.000,C 90.000,E1 160.369} C_DIS
LIN {X -0.019,Y -153.546,Z 1230.871,A 0.000,B 0.000,C 90.000,E1 156.741} C_DIS
LIN {X 0.033,Y -156.963,Z 1230.851,A 0.000,B 0.000,C 90.000,E1 153.127} C_DIS
LIN {X -0.031,Y -161.071,Z 1230.831,A 0.000,B 0.000,C 90.000,E1 149.587} C_DIS
LIN {X 0.053,Y -163.177,Z 1230.821,A 0.000,B 0.000,C 90.000,E1 147.788} C_DIS
LIN {X 0.060,Y -167.599,Z 1230.802,A 0.000,B 0.000,C 90.000,E1 144.276} C_DIS
LIN {X -0.031,Y -171.427,Z 1230.787,A 0.000,B 0.000,C 90.000,E1 141.698} C_DIS
LIN {X 0.008,Y -176.347,Z 1230.768,A 0.000,B 0.000,C 90.000,E1 138.243} C_DIS
LIN {X 0.004,Y -180.637,Z 1230.754,A 0.000,B 0.000,C 90.000,E1 135.688} C_DIS
LIN {X -0.012,Y -186.039,Z 1230.735,A 0.000,B 0.000,C 90.000,E1 132.324} C_DIS
LIN {X 0.051,Y -190.674,Z 1230.721,A 0.000,B 0.000,C 90.000,E1 129.806} C_DIS
LIN {X 0.085,Y -196.426,Z 1230.703,A 0.000,B 0.000,C 90.000,E1 126.503} C_DIS
LIN {X -0.051,Y -200.910,Z 1230.690,A 0.000,B 0.000,C 90.000,E1 124.278} C_DIS
LIN {X 0.061,Y -310.876,Z 1230.690,A 0.000,B 0.000,C 90.000,E1 124.246} C_DIS
LIN {X -0.044,Y -312.177,Z 1230.690,A 0.000,B 0.000,C 90.000,E1 124.246} C_DIS
LIN {X 0.081,Y -316.058,Z 1230.689,A 0.000,B 0.000,C 90.000,E1 124.072} C_DIS
LIN {X 0.050,Y -319.296,Z 1230.688,A 0.000,B 0.000,C 90.000,E1 123.833} C_DIS
LIN {X 0.138,Y -322.977,Z 1230.686,A 0.000,B 0.000,C 90.000,E1 123.372} C_DIS
LIN {X -0.053,Y -324.820,Z 1230.684,A 0.000,B 0.000,C 90.000,E1 123.086} C_DIS
LIN {X 0.027,Y -326.251,Z 1230.682,A 0.000,B 0.000,C 90.000,E1 122.752} C_DIS
LIN {X -0.001,Y -338.209,Z 1230.665,A 0.000,B 0.000,C 90.000,E1 119.617} C_DIS
LIN {X -0.157,Y -350.384,Z 1230.649,A 0.000,B 0.000,C 90.000,E1 116.873} C_DIS
LIN {X 0.014,Y -364.042,Z 1230.634,A 0.000,B 0.000,C 90.000,E1 114.131} C_DIS
LIN {X 0.025,Y -377.519,Z 1230.621,A 0.000,B 0.000,C 90.000,E1 111.770} C_DIS
LIN {X 0.103,Y -392.352,Z 1230.608,A 0.000,B 0.000,C 90.000,E1 109.450} C_DIS
LIN {X -0.078,Y -408.646,Z 1230.596,A 0.000,B 0.000,C 90.000,E1 107.221} C_DIS
LIN {X 0.017,Y -426.517,Z 1230.583,A 0.000,B 0.000,C 90.000,E1 105.009} C_DIS
LIN {X -0.001,Y -445.978,Z 1230.572,A 0.000,B 0.000,C 90.000,E1 102.883} C_DIS
LIN {X 0.143,Y -466.207,Z 1230.561,A 0.000,B 0.000,C 90.000,E1 100.894} C_DIS
LIN {X 0.155,Y -473.736,Z 1230.557,A 0.000,B 0.000,C 90.000,E1 100.197} C_DIS
LIN {X 0.214,Y -475.554,Z 1230.556,A 0.000,B 0.000,C 90.000,E1 99.962} C_DIS
LIN {X 0.079,Y -477.075,Z 1230.554,A 0.000,B 0.000,C 90.000,E1 99.726} C_DIS
LIN {X -0.138,Y -478.212,Z 1230.553,A 0.000,B 0.000,C 90.000,E1 99.500} C_DIS
LIN {X 0.079,Y -479.570,Z 1230.550,A 0.000,B 0.000,C 90.000,E1 98.973} C_DIS
LIN {X 0.227,Y -479.901,Z 1230.547,A 0.000,B 0.000,C 90.000,E1 98.454} C_DIS
LIN {X -0.089,Y -479.261,Z 1230.544,A 0.000,B 0.000,C 90.000,E1 97.992} C_DIS
LIN {X 0.073,Y -477.547,Z 1230.542,A 0.000,B 0.000,C 90.000,E1 97.473} C_DIS
LIN {X -0.054,Y -476.191,Z 1230.540,A 0.000,B 0.000,C 90.000,E1 97.239} C_DIS
LIN {X -0.216,Y -456.221,Z 1230.525,A 0.000,B 0.000,C 90.000,E1 94.473} C_DIS
LIN {X 0.005,Y -435.527,Z 1230.507,A 0.000,B 0.000,C 90.000,E1 91.318} C_DIS
LIN {X -0.122,Y -422.968,Z 1230.495,A 0.000,B 0.000,C 90.000,E1 89.198} C_DIS
LIN {X 0.146,Y -407.057,Z 1230.479,A 0.000,B 0.000,C 90.000,E1 86.159} C_DIS
LIN {X -0.195,Y -396.938,Z 1230.468,A 0.000,B 0.000,C 90.000,E1 84.261} C_DIS
LIN {X 0.082,Y -386.748,Z 1230.457,A 0.000,B 0.000,C 90.000,E1 82.243} C_DIS
LIN {X -0.146,Y -377.870,Z 1230.447,A 0.000,B 0.000,C 90.000,E1 80.557} C_DIS
LIN {X -0.155,Y -368.685,Z 1230.438,A 0.000,B 0.000,C 90.000,E1 78.814} C_DIS
LIN {X 0.166,Y -359.293,Z 1230.428,A 0.000,B 0.000,C 90.000,E1 76.992} C_DIS
LIN {X -0.039,Y -349.637,Z 1230.418,A 0.000,B 0.000,C 90.000,E1 75.227} C_DIS
LIN {X -0.005,Y -336.717,Z 1230.404,A 0.000,B 0.000,C 90.000,E1 72.779} C_DIS
LIN {X -0.037,Y -325.629,Z 1230.392,A 0.000,B 0.000,C 90.000,E1 70.604} C_DIS
LIN {X -0.088,Y -309.040,Z 1230.373,A 0.000,B 0.000,C 90.000,E1 67.102} C_DIS
LIN {X 0.068,Y -293.923,Z 1230.353,A 0.000,B 0.000,C 90.000,E1 63.461} C_DIS
LIN {X -0.111,Y -281.318,Z 1230.334,A 0.000,B 0.000,C 90.000,E1 60.127} C_DIS
LIN {X 0.140,Y -269.743,Z 1230.315,A 0.000,B 0.000,C 90.000,E1 56.628} C_DIS
LIN {X 0.046,Y -259.066,Z 1230.295,A 0.000,B 0.000,C 90.000,E1 53.130} C_DIS
LIN {X 0.051,Y -249.276,Z 1230.275,A 0.000,B 0.000,C 90.000,E1 49.542} C_DIS
LIN {X 0.027,Y -240.169,Z 1230.255,A 0.000,B 0.000,C 90.000,E1 45.891} C_DIS
LIN {X -0.031,Y -233.204,Z 1230.239,A 0.000,B 0.000,C 90.000,E1 42.933} C_DIS
LIN {X -0.079,Y -226.422,Z 1230.222,A 0.000,B 0.000,C 90.000,E1 39.930} C_DIS
LIN {X -0.033,Y -218.526,Z 1230.200,A 0.000,B 0.000,C 90.000,E1 36.091} C_DIS
LIN {X -0.078,Y -211.497,Z 1230.179,A 0.000,B 0.000,C 90.000,E1 32.212} C_DIS
LIN {X 0.041,Y -205.391,Z 1230.157,A 0.000,B 0.000,C 90.000,E1 28.231} C_DIS
LIN {X -0.058,Y -200.205,Z 1230.135,A 0.000,B 0.000,C 90.000,E1 24.259} C_DIS
LIN {X 0.018,Y -196.000,Z 1230.112,A 0.000,B 0.000,C 90.000,E1 20.194} C_DIS
LIN {X -0.003,Y -192.002,Z 1230.085,A 0.000,B 0.000,C 90.000,E1 15.300} C_DIS
LIN {X -0.079,Y -188.937,Z 1230.053,A 0.000,B 0.000,C 90.000,E1 9.557} C_DIS
LIN {X -0.034,Y -190.033,Z 1229.965,A 0.000,B 0.000,C 90.000,E1 353.742} C_DIS
LIN {X -0.094,Y -193.129,Z 1229.938,A 0.000,B 0.000,C 90.000,E1 348.814} C_DIS
LIN {X 0.040,Y -197.372,Z 1229.910,A 0.000,B 0.000,C 90.000,E1 343.866} C_DIS
LIN {X -0.007,Y -201.840,Z 1229.888,A 0.000,B 0.000,C 90.000,E1 339.826} C_DIS
LIN {X 0.067,Y -207.056,Z 1229.866,A 0.000,B 0.000,C 90.000,E1 335.793} C_DIS
LIN {X -0.003,Y -212.924,Z 1229.844,A 0.000,B 0.000,C 90.000,E1 331.847} C_DIS
LIN {X 0.057,Y -219.220,Z 1229.822,A 0.000,B 0.000,C 90.000,E1 327.916} C_DIS
LIN {X -0.005,Y -226.260,Z 1229.800,A 0.000,B 0.000,C 90.000,E1 324.069} C_DIS
LIN {X -0.048,Y -233.969,Z 1229.779,A 0.000,B 0.000,C 90.000,E1 320.275} C_DIS
LIN {X -0.083,Y -242.584,Z 1229.758,A 0.000,B 0.000,C 90.000,E1 316.539} C_DIS
LIN {X -0.031,Y -249.448,Z 1229.744,A 0.000,B 0.000,C 90.000,E1 313.947} C_DIS
LIN {X 0.035,Y -257.175,Z 1229.730,A 0.000,B 0.000,C 90.000,E1 311.391} C_DIS
LIN {X -0.057,Y -266.011,Z 1229.716,A 0.000,B 0.000,C 90.000,E1 308.910} C_DIS
LIN {X -0.005,Y -274.479,Z 1229.704,A 0.000,B 0.000,C 90.000,E1 306.790} C_DIS
LIN {X -0.048,Y -287.108,Z 1229.689,A 0.000,B 0.000,C 90.000,E1 304.040} C_DIS
LIN {X -0.010,Y -299.478,Z 1229.676,A 0.000,B 0.000,C 90.000,E1 301.671} C_DIS
LIN {X 0.053,Y -307.020,Z 1229.669,A 0.000,B 0.000,C 90.000,E1 300.335} C_DIS
LIN {X 0.062,Y -315.614,Z 1229.661,A 0.000,B 0.000,C 90.000,E1 299.027} C_DIS
LIN {X -0.056,Y -330.355,Z 1229.651,A 0.000,B 0.000,C 90.000,E1 297.129} C_DIS
LIN {X 0.013,Y -351.369,Z 1229.637,A 0.000,B 0.000,C 90.000,E1 294.643} C_DIS
LIN {X 0.030,Y -375.271,Z 1229.622,A 0.000,B 0.000,C 90.000,E1 292.025} C_DIS
LIN {X 0.179,Y -388.374,Z 1229.615,A 0.000,B 0.000,C 90.000,E1 290.610} C_DIS
LIN {X 0.078,Y -406.478,Z 1229.604,A 0.000,B 0.000,C 90.000,E1 288.725} C_DIS
LIN {X -0.034,Y -416.615,Z 1229.598,A 0.000,B 0.000,C 90.000,E1 287.692} C_DIS
LIN {X -0.179,Y -424.049,Z 1229.594,A 0.000,B 0.000,C 90.000,E1 286.913} C_DIS
LIN {X -0.017,Y -431.134,Z 1229.589,A 0.000,B 0.000,C 90.000,E1 286.079} C_DIS
LIN {X 0.210,Y -437.666,Z 1229.585,A 0.000,B 0.000,C 90.000,E1 285.245} C_DIS
LIN {X -0.033,Y -443.604,Z 1229.580,A 0.000,B 0.000,C 90.000,E1 284.481} C_DIS
LIN {X -0.125,Y -448.885,Z 1229.576,A 0.000,B 0.000,C 90.000,E1 283.703} C_DIS
LIN {X 0.167,Y -453.509,Z 1229.572,A 0.000,B 0.000,C 90.000,E1 282.883} C_DIS
LIN {X 0.055,Y -457.441,Z 1229.567,A 0.000,B 0.000,C 90.000,E1 282.119} C_DIS
LIN {X 0.150,Y -459.726,Z 1229.564,A 0.000,B 0.000,C 90.000,E1 281.591} C_DIS
LIN {X 0.170,Y -461.701,Z 1229.562,A 0.000,B 0.000,C 90.000,E1 281.074} C_DIS
LIN {X -0.167,Y -463.426,Z 1229.559,A 0.000,B 0.000,C 90.000,E1 280.602} C_DIS
LIN {X -0.042,Y -464.866,Z 1229.556,A 0.000,B 0.000,C 90.000,E1 280.074} C_DIS
LIN {X 0.013,Y -466.050,Z 1229.553,A 0.000,B 0.000,C 90.000,E1 279.557} C_DIS
LIN {X 0.155,Y -467.020,Z 1229.550,A 0.000,B 0.000,C 90.000,E1 279.029} C_DIS
LIN {X 0.230,Y -467.643,Z 1229.547,A 0.000,B 0.000,C 90.000,E1 278.511} C_DIS
LIN {X -0.151,Y -467.980,Z 1229.545,A 0.000,B 0.000,C 90.000,E1 278.049} C_DIS
LIN {X -0.062,Y -467.976,Z 1229.542,A 0.000,B 0.000,C 90.000,E1 277.530} C_DIS
LIN {X 0.087,Y -467.611,Z 1229.539,A 0.000,B 0.000,C 90.000,E1 277.004} C_DIS
LIN {X 0.175,Y -466.809,Z 1229.536,A 0.000,B 0.000,C 90.000,E1 276.486} C_DIS
LIN {X -0.202,Y -465.599,Z 1229.533,A 0.000,B 0.000,C 90.000,E1 276.024} C_DIS
LIN {X -0.166,Y -463.951,Z 1229.531,A 0.000,B 0.000,C 90.000,E1 275.511} C_DIS
LIN {X -0.089,Y -461.883,Z 1229.528,A 0.000,B 0.000,C 90.000,E1 274.992} C_DIS
LIN {X -0.024,Y -459.339,Z 1229.525,A 0.000,B 0.000,C 90.000,E1 274.473} C_DIS
LIN {X 0.019,Y -456.128,Z 1229.522,A 0.000,B 0.000,C 90.000,E1 273.955} C_DIS
LIN {X -0.210,Y -454.258,Z 1229.521,A 0.000,B 0.000,C 90.000,E1 273.726} C_DIS
LIN {X -0.219,Y -449.715,Z 1229.518,A 0.000,B 0.000,C 90.000,E1 273.212} C_DIS
LIN {X -0.100,Y -444.124,Z 1229.515,A 0.000,B 0.000,C 90.000,E1 272.694} C_DIS
LIN {X -0.038,Y -437.837,Z 1229.512,A 0.000,B 0.000,C 90.000,E1 272.236} C_DIS
LIN {X 0.128,Y -431.072,Z 1229.510,A 0.000,B 0.000,C 90.000,E1 271.835} C_DIS
LIN {X -0.094,Y -423.971,Z 1229.509,A 0.000,B 0.000,C 90.000,E1 271.547} C_DIS
LIN {X 0.065,Y -416.893,Z 1229.507,A 0.000,B 0.000,C 90.000,E1 271.260} C_DIS
LIN {X 0.120,Y -409.799,Z 1229.506,A 0.000,B 0.000,C 90.000,E1 271.031} C_DIS
LIN {X -0.163,Y -398.986,Z 1229.504,A 0.000,B 0.000,C 90.000,E1 270.802} C_DIS
LIN {X -0.044,Y -388.300,Z 1229.503,A 0.000,B 0.000,C 90.000,E1 270.573} C_DIS
LIN {X -0.013,Y -379.078,Z 1229.503,A 0.000,B 0.000,C 90.000,E1 270.458} C_DIS
LIN {X -0.068,Y -370.446,Z 1229.502,A 0.000,B 0.000,C 90.000,E1 270.401} C_DIS
LIN {X 0.180,Y -365.541,Z 1229.502,A 0.000,B 0.000,C 90.000,E1 270.344} C_DIS
LIN {X 0.060,Y -181.579,Z 1229.502,A 0.000,B 0.000,C 90.000,E1 270.344} C_DIS
LIN {X -0.015,Y -180.849,Z 1229.472,A 0.000,B 0.000,C 90.000,E1 264.951} C_DIS
LIN {X 0.067,Y -178.958,Z 1229.444,A 0.000,B 0.000,C 90.000,E1 259.859} C_DIS
LIN {X -0.042,Y -177.363,Z 1229.430,A 0.000,B 0.000,C 90.000,E1 257.353} C_DIS
LIN {X 0.054,Y -175.535,Z 1229.411,A 0.000,B 0.000,C 90.000,E1 253.921} C_DIS
LIN {X 0.055,Y -172.270,Z 1229.387,A 0.000,B 0.000,C 90.000,E1 249.645} C_DIS
LIN {X 0.094,Y -171.748,Z 1229.382,A 0.000,B 0.000,C 90.000,E1 248.773} C_DIS
LIN {X -0.048,Y -167.347,Z 1229.354,A 0.000,B 0.000,C 90.000,E1 243.640} C_DIS
LIN {X 0.033,Y -166.733,Z 1229.349,A 0.000,B 0.000,C 90.000,E1 242.743} C_DIS
LIN {X -0.055,Y -162.714,Z 1229.324,A 0.000,B 0.000,C 90.000,E1 238.408} C_DIS
LIN {X 0.008,Y -161.404,Z 1229.315,A 0.000,B 0.000,C 90.000,E1 236.628} C_DIS
LIN {X 0.049,Y -157.397,Z 1229.290,A 0.000,B 0.000,C 90.000,E1 232.190} C_DIS
LIN {X -0.018,Y -155.395,Z 1229.275,A 0.000,B 0.000,C 90.000,E1 229.542} C_DIS
LIN {X 0.021,Y -151.728,Z 1229.250,A 0.000,B 0.000,C 90.000,E1 225.040} C_DIS
LIN {X -0.074,Y -149.923,Z 1229.235,A 0.000,B 0.000,C 90.000,E1 222.366} C_DIS
LIN {X -0.046,Y -146.775,Z 1229.210,A 0.000,B 0.000,C 90.000,E1 217.810} C_DIS
LIN {X 0.058,Y -145.345,Z 1229.195,A 0.000,B 0.000,C 90.000,E1 215.025} C_DIS
LIN {X -0.027,Y -142.420,Z 1229.164,A 0.000,B 0.000,C 90.000,E1 209.539} C_DIS
LIN {X 0.024,Y -141.407,Z 1229.149,A 0.000,B 0.000,C 90.000,E1 206.744} C_DIS
LIN {X 0.011,Y -139.357,Z 1229.113,A 0.000,B 0.000,C 90.000,E1 200.248} C_DIS
LIN {X -0.001,Y -138.799,Z 1229.097,A 0.000,B 0.000,C 90.000,E1 197.457} C_DIS
LIN {X 0.053,Y -138.348,Z 1229.055,A 0.000,B 0.000,C 90.000,E1 189.962} C_DIS
LIN {X 0.071,Y -139.370,Z 1229.009,A 0.000,B 0.000,C 90.000,E1 181.547} C_DIS
LIN {X -0.015,Y -141.258,Z 1228.973,A 0.000,B 0.000,C 90.000,E1 175.065} C_DIS
LIN {X -0.058,Y -142.626,Z 1228.957,A 0.000,B 0.000,C 90.000,E1 172.299} C_DIS
LIN {X 0.036,Y -144.948,Z 1228.931,A 0.000,B 0.000,C 90.000,E1 167.645} C_DIS
LIN {X 0.027,Y -147.576,Z 1228.911,A 0.000,B 0.000,C 90.000,E1 163.976} C_DIS
LIN {X -0.084,Y -150.189,Z 1228.891,A 0.000,B 0.000,C 90.000,E1 160.369} C_DIS
LIN {X -0.076,Y -153.567,Z 1228.871,A 0.000,B 0.000,C 90.000,E1 156.741} C_DIS
LIN {X -0.025,Y -156.984,Z 1228.851,A 0.000,B 0.000,C 90.000,E1 153.127} C_DIS
LIN {X 0.048,Y -161.097,Z 1228.831,A 0.000,B 0.000,C 90.000,E1 149.537} C_DIS
LIN {X -0.006,Y -163.202,Z 1228.821,A 0.000,B 0.000,C 90.000,E1 147.788} C_DIS
LIN {X -0.001,Y -167.628,Z 1228.802,A 0.000,B 0.000,C 90.000,E1 144.276} C_DIS
LIN {X 0.014,Y -171.454,Z 1228.787,A 0.000,B 0.000,C 90.000,E1 141.662} C_DIS
LIN {X -0.055,Y -176.379,Z 1228.768,A 0.000,B 0.000,C 90.000,E1 138.243} C_DIS
LIN {X 0.067,Y -180.671,Z 1228.754,A 0.000,B 0.000,C 90.000,E1 135.648} C_DIS
LIN {X 0.049,Y -186.074,Z 1228.735,A 0.000,B 0.000,C 90.000,E1 132.285} C_DIS
LIN {X -0.014,Y -190.710,Z 1228.721,A 0.000,B 0.000,C 90.000,E1 129.806} C_DIS
LIN {X 0.018,Y -196.462,Z 1228.703,A 0.000,B 0.000,C 90.000,E1 126.503} C_DIS
LIN {X -0.029,Y -200.955,Z 1228.690,A 0.000,B 0.000,C 90.000,E1 124.246} C_DIS
LIN {X -0.079,Y -311.142,Z 1228.690,A 0.000,B 0.000,C 90.000,E1 124.246} C_DIS
LIN {X -0.025,Y -316.049,Z 1228.689,A 0.000,B 0.000,C 90.000,E1 124.072} C_DIS
LIN {X -0.007,Y -319.223,Z 1228.688,A 0.000,B 0.000,C 90.000,E1 123.833} C_DIS
LIN {X 0.117,Y -322.913,Z 1228.686,A 0.000,B 0.000,C 90.000,E1 123.372} C_DIS
LIN {X -0.058,Y -324.768,Z 1228.684,A 0.000,B 0.000,C 90.000,E1 123.086} C_DIS
LIN {X 0.041,Y -326.211,Z 1228.682,A 0.000,B 0.000,C 90.000,E1 122.752} C_DIS
LIN {X 0.011,Y -338.178,Z 1228.665,A 0.000,B 0.000,C 90.000,E1 119.617} C_DIS
LIN {X -0.145,Y -350.353,Z 1228.649,A 0.000,B 0.000,C 90.000,E1 116.873} C_DIS
LIN {X 0.027,Y -364.009,Z 1228.634,A 0.000,B 0.000,C 90.000,E1 114.131} C_DIS
LIN {X 0.037,Y -377.484,Z 1228.621,A 0.000,B 0.000,C 90.000,E1 111.770} C_DIS
LIN {X 0.113,Y -392.315,Z 1228.608,A 0.000,B 0.000,C 90.000,E1 109.450} C_DIS
LIN {X -0.068,Y -408.608,Z 1228.596,A 0.000,B 0.000,C 90.000,E1 107.221} C_DIS
LIN {X 0.027,Y -426.478,Z 1228.583,A 0.000,B 0.000,C 90.000,E1 105.009} C_DIS
LIN {X 0.009,Y -445.938,Z 1228.572,A 0.000,B 0.000,C 90.000,E1 102.883} C_DIS
LIN {X 0.151,Y -466.167,Z 1228.561,A 0.000,B 0.000,C 90.000,E1 100.894} C_DIS
LIN {X 0.163,Y -473.681,Z 1228.557,A 0.000,B 0.000,C 90.000,E1 100.197} C_DIS
LIN {X 0.221,Y -475.483,Z 1228.556,A 0.000,B 0.000,C 90.000,E1 99.962} C_DIS
LIN {X 0.086,Y -476.991,Z 1228.554,A 0.000,B 0.000,C 90.000,E1 99.726} C_DIS
LIN {X -0.130,Y -478.119,Z 1228.553,A 0.000,B 0.000,C 90.000,E1 99.500} C_DIS
LIN {X 0.086,Y -479.461,Z 1228.550,A 0.000,B 0.000,C 90.000,E1 98.973} C_DIS
LIN {X -0.241,Y -479.779,Z 1228.547,A 0.000,B 0.000,C 90.000,E1 98.511} C_DIS
LIN {X -0.083,Y -479.124,Z 1228.544,A 0.000,B 0.000,C 90.000,E1 97.992} C_DIS
LIN {X 0.078,Y -477.394,Z 1228.542,A 0.000,B 0.000,C 90.000,E1 97.473} C_DIS
LIN {X -0.050,Y -476.028,Z 1228.540,A 0.000,B 0.000,C 90.000,E1 97.239} C_DIS
LIN {X -0.216,Y -456.042,Z 1228.525,A 0.000,B 0.000,C 90.000,E1 94.473} C_DIS
LIN {X -0.002,Y -435.366,Z 1228.507,A 0.000,B 0.000,C 90.000,E1 91.318} C_DIS
LIN {X -0.131,Y -422.817,Z 1228.495,A 0.000,B 0.000,C 90.000,E1 89.198} C_DIS
LIN {X 0.064,Y -408.305,Z 1228.480,A 0.000,B 0.000,C 90.000,E1 86.445} C_DIS
LIN {X 0.147,Y -398.217,Z 1228.469,A 0.000,B 0.000,C 90.000,E1 84.489} C_DIS
LIN {X 0.018,Y -388.036,Z 1228.458,A 0.000,B 0.000,C 90.000,E1 82.534} C_DIS
LIN {X 0.183,Y -379.187,Z 1228.449,A 0.000,B 0.000,C 90.000,E1 80.792} C_DIS
LIN {X -0.176,Y -370.089,Z 1228.439,A 0.000,B 0.000,C 90.000,E1 79.106} C_DIS
LIN {X 0.092,Y -360.712,Z 1228.430,A 0.000,B 0.000,C 90.000,E1 77.297} C_DIS
LIN {X -0.069,Y -349.468,Z 1228.418,A 0.000,B 0.000,C 90.000,E1 75.227} C_DIS
LIN {X -0.031,Y -338.175,Z 1228.406,A 0.000,B 0.000,C 90.000,E1 73.087} C_DIS
LIN {X -0.041,Y -327.062,Z 1228.394,A 0.000,B 0.000,C 90.000,E1 70.913} C_DIS
LIN {X -0.042,Y -310.354,Z 1228.375,A 0.000,B 0.000,C 90.000,E1 67.411} C_DIS
LIN {X 0.155,Y -295.105,Z 1228.354,A 0.000,B 0.000,C 90.000,E1 63.768} C_DIS
LIN {X -0.123,Y -282.381,Z 1228.336,A 0.000,B 0.000,C 90.000,E1 60.461} C_DIS
LIN {X 0.013,Y -270.668,Z 1228.317,A 0.000,B 0.000,C 90.000,E1 56.993} C_DIS
LIN {X 0.040,Y -260.928,Z 1228.299,A 0.000,B 0.000,C 90.000,E1 53.829} C_DIS
LIN {X -0.048,Y -250.924,Z 1228.279,A 0.000,B 0.000,C 90.000,E1 50.275} C_DIS
LIN {X 0.000,Y -241.649,Z 1228.259,A 0.000,B 0.000,C 90.000,E1 46.620} C_DIS
LIN {X -0.024,Y -234.599,Z 1228.243,A 0.000,B 0.000,C 90.000,E1 43.662} C_DIS
LIN {X 0.119,Y -227.721,Z 1228.226,A 0.000,B 0.000,C 90.000,E1 40.620} C_DIS
LIN {X 0.028,Y -219.648,Z 1228.205,A 0.000,B 0.000,C 90.000,E1 36.824} C_DIS
LIN {X -0.036,Y -212.426,Z 1228.183,A 0.000,B 0.000,C 90.000,E1 32.959} C_DIS
LIN {X 0.035,Y -206.139,Z 1228.161,A 0.000,B 0.000,C 90.000,E1 28.999} C_DIS
LIN {X -0.041,Y -200.798,Z 1228.139,A 0.000,B 0.000,C 90.000,E1 25.027} C_DIS
LIN {X 0.017,Y -196.431,Z 1228.117,A 0.000,B 0.000,C 90.000,E1 20.972} C_DIS
LIN {X 0.007,Y -192.250,Z 1228.089,A 0.000,B 0.000,C 90.000,E1 16.079} C_DIS
LIN {X 0.023,Y -188.941,Z 1228.057,A 0.000,B 0.000,C 90.000,E1 10.310} C_DIS
LIN {X -0.048,Y -189.723,Z 1227.965,A 0.000,B 0.000,C 90.000,E1 353.742} C_DIS
LIN {X 0.069,Y -192.817,Z 1227.938,A 0.000,B 0.000,C 90.000,E1 348.757} C_DIS
LIN {X 0.002,Y -197.090,Z 1227.910,A 0.000,B 0.000,C 90.000,E1 343.866} C_DIS
LIN {X -0.055,Y -201.582,Z 1227.888,A 0.000,B 0.000,C 90.000,E1 339.826} C_DIS
LIN {X 0.010,Y -206.833,Z 1227.865,A 0.000,B 0.000,C 90.000,E1 335.793} C_DIS
LIN {X -0.068,Y -212.722,Z 1227.844,A 0.000,B 0.000,C 90.000,E1 331.847} C_DIS
LIN {X -0.016,Y -219.043,Z 1227.822,A 0.000,B 0.000,C 90.000,E1 327.916} C_DIS
LIN {X -0.086,Y -226.101,Z 1227.800,A 0.000,B 0.000,C 90.000,E1 324.069} C_DIS
LIN {X 0.042,Y -233.812,Z 1227.779,A 0.000,B 0.000,C 90.000,E1 320.231} C_DIS
LIN {X -0.014,Y -242.443,Z 1227.758,A 0.000,B 0.000,C 90.000,E1 316.500} C_DIS
LIN {X 0.046,Y -248.289,Z 1227.746,A 0.000,B 0.000,C 90.000,E1 314.271} C_DIS
LIN {X -0.074,Y -257.102,Z 1227.730,A 0.000,B 0.000,C 90.000,E1 311.391} C_DIS
LIN {X -0.005,Y -265.998,Z 1227.716,A 0.000,B 0.000,C 90.000,E1 308.874} C_DIS
LIN {X -0.123,Y -274.459,Z 1227.704,A 0.000,B 0.000,C 90.000,E1 306.790} C_DIS
LIN {X 0.067,Y -287.110,Z 1227.689,A 0.000,B 0.000,C 90.000,E1 303.992} C_DIS
LIN {X -0.130,Y -301.301,Z 1227.674,A 0.000,B 0.000,C 90.000,E1 301.337} C_DIS
LIN {X -0.047,Y -308.986,Z 1227.667,A 0.000,B 0.000,C 90.000,E1 300.001} C_DIS
LIN {X 0.078,Y -315.520,Z 1227.661,A 0.000,B 0.000,C 90.000,E1 298.999} C_DIS
LIN {X -0.113,Y -330.124,Z 1227.651,A 0.000,B 0.000,C 90.000,E1 297.129} C_DIS
LIN {X -0.086,Y -348.573,Z 1227.639,A 0.000,B 0.000,C 90.000,E1 294.951} C_DIS
LIN {X -0.140,Y -372.381,Z 1227.624,A 0.000,B 0.000,C 90.000,E1 292.333} C_DIS
LIN {X 0.065,Y -385.448,Z 1227.616,A 0.000,B 0.000,C 90.000,E1 290.918} C_DIS
LIN {X 0.162,Y -401.009,Z 1227.607,A 0.000,B 0.000,C 90.000,E1 289.268} C_DIS
LIN {X 0.118,Y -413.928,Z 1227.600,A 0.000,B 0.000,C 90.000,E1 287.946} C_DIS
LIN {X -0.011,Y -421.482,Z 1227.595,A 0.000,B 0.000,C 90.000,E1 287.166} C_DIS
LIN {X -0.115,Y -428.707,Z 1227.591,A 0.000,B 0.000,C 90.000,E1 286.370} C_DIS
LIN {X -0.026,Y -435.452,Z 1227.586,A 0.000,B 0.000,C 90.000,E1 285.552} C_DIS
LIN {X -0.183,Y -441.602,Z 1227.582,A 0.000,B 0.000,C 90.000,E1 284.773} C_DIS
LIN {X 0.038,Y -447.125,Z 1227.578,A 0.000,B 0.000,C 90.000,E1 283.953} C_DIS
LIN {X -0.023,Y -451.996,Z 1227.573,A 0.000,B 0.000,C 90.000,E1 283.175} C_DIS
LIN {X -0.145,Y -456.209,Z 1227.569,A 0.000,B 0.000,C 90.000,E1 282.411} C_DIS
LIN {X 0.213,Y -459.743,Z 1227.565,A 0.000,B 0.000,C 90.000,E1 281.591} C_DIS
LIN {X -0.220,Y -461.736,Z 1227.562,A 0.000,B 0.000,C 90.000,E1 281.130} C_DIS
LIN {X -0.104,Y -463.469,Z 1227.559,A 0.000,B 0.000,C 90.000,E1 280.602} C_DIS
LIN {X 0.022,Y -464.936,Z 1227.556,A 0.000,B 0.000,C 90.000,E1 280.074} C_DIS
LIN {X 0.078,Y -466.122,Z 1227.553,A 0.000,B 0.000,C 90.000,E1 279.557} C_DIS
LIN {X 0.220,Y -467.062,Z 1227.550,A 0.000,B 0.000,C 90.000,E1 279.029} C_DIS
LIN {X -0.167,Y -467.729,Z 1227.547,A 0.000,B 0.000,C 90.000,E1 278.568} C_DIS
LIN {X -0.084,Y -468.084,Z 1227.545,A 0.000,B 0.000,C 90.000,E1 278.049} C_DIS
LIN {X 0.004,Y -468.104,Z 1227.542,A 0.000,B 0.000,C 90.000,E1 277.530} C_DIS
LIN {X 0.097,Y -467.746,Z 1227.539,A 0.000,B 0.000,C 90.000,E1 277.011} C_DIS
LIN {X 0.243,Y -466.973,Z 1227.536,A 0.000,B 0.000,C 90.000,E1 276.486} C_DIS
LIN {X -0.134,Y -465.788,Z 1227.533,A 0.000,B 0.000,C 90.000,E1 276.024} C_DIS
LIN {X -0.097,Y -464.186,Z 1227.531,A 0.000,B 0.000,C 90.000,E1 275.511} C_DIS
LIN {X -0.196,Y -460.960,Z 1227.526,A 0.000,B 0.000,C 90.000,E1 274.759} C_DIS
LIN {X -0.176,Y -458.135,Z 1227.523,A 0.000,B 0.000,C 90.000,E1 274.245} C_DIS
LIN {X -0.137,Y -454.585,Z 1227.521,A 0.000,B 0.000,C 90.000,E1 273.726} C_DIS
LIN {X -0.146,Y -450.102,Z 1227.518,A 0.000,B 0.000,C 90.000,E1 273.212} C_DIS
LIN {X 0.092,Y -447.422,Z 1227.516,A 0.000,B 0.000,C 90.000,E1 272.922} C_DIS
LIN {X -0.176,Y -441.291,Z 1227.514,A 0.000,B 0.000,C 90.000,E1 272.465} C_DIS
LIN {X -0.036,Y -438.194,Z 1227.512,A 0.000,B 0.000,C 90.000,E1 272.236} C_DIS
LIN {X 0.093,Y -431.393,Z 1227.510,A 0.000,B 0.000,C 90.000,E1 271.835} C_DIS
LIN {X -0.114,Y -424.324,Z 1227.509,A 0.000,B 0.000,C 90.000,E1 271.547} C_DIS
LIN {X 0.068,Y -417.346,Z 1227.507,A 0.000,B 0.000,C 90.000,E1 271.260} C_DIS
LIN {X 0.139,Y -410.353,Z 1227.506,A 0.000,B 0.000,C 90.000,E1 271.031} C_DIS
LIN {X -0.175,Y -399.604,Z 1227.504,A 0.000,B 0.000,C 90.000,E1 270.802} C_DIS
LIN {X -0.073,Y -388.867,Z 1227.503,A 0.000,B 0.000,C 90.000,E1 270.573} C_DIS
LIN {X -0.064,Y -380.008,Z 1227.502,A 0.000,B 0.000,C 90.000,E1 270.458} C_DIS
LIN {X 0.107,Y -367.494,Z 1227.502,A 0.000,B 0.000,C 90.000,E1 270.344} C_DIS
LIN {X 0.047,Y -364.479,Z 1227.502,A 0.000,B 0.000,C 90.000,E1 270.344} C_DIS
LIN {X -0.006,Y -181.579,Z 1227.502,A 0.000,B 0.000,C 90.000,E1 270.344} C_DIS
LIN {X -0.053,Y -180.845,Z 1227.472,A 0.000,B 0.000,C 90.000,E1 264.951} C_DIS
LIN {X 0.030,Y -178.954,Z 1227.444,A 0.000,B 0.000,C 90.000,E1 259.859} C_DIS
LIN {X -0.078,Y -177.356,Z 1227.430,A 0.000,B 0.000,C 90.000,E1 257.353} C_DIS
LIN {X 0.017,Y -175.526,Z 1227.411,A 0.000,B 0.000,C 90.000,E1 253.921} C_DIS
LIN {X 0.019,Y -172.262,Z 1227.387,A 0.000,B 0.000,C 90.000,E1 249.645} C_DIS
LIN {X 0.057,Y -171.741,Z 1227.382,A 0.000,B 0.000,C 90.000,E1 248.773} C_DIS
LIN {X -0.084,Y -167.338,Z 1227.353,A 0.000,B 0.000,C 90.000,E1 243.640} C_DIS
LIN {X -0.002,Y -166.724,Z 1227.349,A 0.000,B 0.000,C 90.000,E1 242.743} C_DIS
LIN {X -0.089,Y -162.704,Z 1227.324,A 0.000,B 0.000,C 90.000,E1 238.408} C_DIS
LIN {X -0.027,Y -161.395,Z 1227.315,A 0.000,B 0.000,C 90.000,E1 236.628} C_DIS
LIN {X 0.015,Y -157.388,Z 1227.290,A 0.000,B 0.000,C 90.000,E1 232.190} C_DIS
LIN {X -0.052,Y -155.383,Z 1227.275,A 0.000,B 0.000,C 90.000,E1 229.542} C_DIS
LIN {X -0.012,Y -151.719,Z 1227.250,A 0.000,B 0.000,C 90.000,E1 225.040} C_DIS
LIN {X 0.004,Y -149.912,Z 1227.235,A 0.000,B 0.000,C 90.000,E1 222.324} C_DIS
LIN {X -0.078,Y -146.768,Z 1227.210,A 0.000,B 0.000,C 90.000,E1 217.810} C_DIS
LIN {X 0.026,Y -145.337,Z 1227.195,A 0.000,B 0.000,C 90.000,E1 215.025} C_DIS
LIN {X -0.059,Y -142.416,Z 1227.164,A 0.000,B 0.000,C 90.000,E1 209.539} C_DIS
LIN {X -0.009,Y -141.401,Z 1227.149,A 0.000,B 0.000,C 90.000,E1 206.744} C_DIS
LIN {X -0.021,Y -139.355,Z 1227.112,A 0.000,B 0.000,C 90.000,E1 200.248} C_DIS
LIN {X -0.033,Y -138.796,Z 1227.097,A 0.000,B 0.000,C 90.000,E1 197.457} C_DIS
LIN {X 0.021,Y -138.347,Z 1227.055,A 0.000,B 0.000,C 90.000,E1 189.962} C_DIS
LIN {X 0.039,Y -139.374,Z 1227.009,A 0.000,B 0.000,C 90.000,E1 181.547} C_DIS
LIN {X -0.048,Y -141.264,Z 1226.973,A 0.000,B 0.000,C 90.000,E1 175.065} C_DIS
LIN {X 0.052,Y -142.630,Z 1226.957,A 0.000,B 0.000,C 90.000,E1 172.243} C_DIS
LIN {X 0.003,Y -144.956,Z 1226.931,A 0.000,B 0.000,C 90.000,E1 167.645} C_DIS
LIN {X -0.006,Y -147.585,Z 1226.911,A 0.000,B 0.000,C 90.000,E1 163.976} C_DIS
LIN {X 0.024,Y -150.198,Z 1226.891,A 0.000,B 0.000,C 90.000,E1 160.315} C_DIS
LIN {X 0.092,Y -153.581,Z 1226.871,A 0.000,B 0.000,C 90.000,E1 156.666} C_DIS
LIN {X -0.059,Y -156.997,Z 1226.851,A 0.000,B 0.000,C 90.000,E1 153.127} C_DIS
LIN {X 0.013,Y -161.113,Z 1226.831,A 0.000,B 0.000,C 90.000,E1 149.537} C_DIS
LIN {X -0.041,Y -163.216,Z 1226.821,A 0.000,B 0.000,C 90.000,E1 147.788} C_DIS
LIN {X -0.037,Y -167.645,Z 1226.802,A 0.000,B 0.000,C 90.000,E1 144.276} C_DIS
LIN {X -0.022,Y -171.470,Z 1226.787,A 0.000,B 0.000,C 90.000,E1 141.662} C_DIS
LIN {X -0.092,Y -176.397,Z 1226.768,A 0.000,B 0.000,C 90.000,E1 138.243} C_DIS
LIN {X 0.029,Y -180.691,Z 1226.754,A 0.000,B 0.000,C 90.000,E1 135.648} C_DIS
LIN {X 0.012,Y -186.094,Z 1226.735,A 0.000,B 0.000,C 90.000,E1 132.285} C_DIS
LIN {X -0.052,Y -190.731,Z 1226.721,A 0.000,B 0.000,C 90.000,E1 129.806} C_DIS
LIN {X -0.021,Y -196.485,Z 1226.703,A 0.000,B 0.000,C 90.000,E1 126.503} C_DIS
LIN {X 0.074,Y -200.986,Z 1226.690,A 0.000,B 0.000,C 90.000,E1 124.199} C_DIS
LIN {X 0.078,Y -310.390,Z 1226.690,A 0.000,B 0.000,C 90.000,E1 124.199} C_DIS
LIN {X -0.087,Y -315.879,Z 1226.689,A 0.000,B 0.000,C 90.000,E1 124.072} C_DIS
LIN {X 0.093,Y -318.810,Z 1226.688,A 0.000,B 0.000,C 90.000,E1 123.833} C_DIS
LIN {X 0.061,Y -322.547,Z 1226.686,A 0.000,B 0.000,C 90.000,E1 123.420} C_DIS
LIN {X 0.054,Y -324.433,Z 1226.684,A 0.000,B 0.000,C 90.000,E1 123.118} C_DIS
LIN {X -0.048,Y -325.910,Z 1226.682,A 0.000,B 0.000,C 90.000,E1 122.832} C_DIS
LIN {X 0.059,Y -339.180,Z 1226.663,A 0.000,B 0.000,C 90.000,E1 119.361} C_DIS
LIN {X -0.070,Y -351.484,Z 1226.648,A 0.000,B 0.000,C 90.000,E1 116.616} C_DIS
LIN {X -0.008,Y -365.273,Z 1226.633,A 0.000,B 0.000,C 90.000,E1 113.898} C_DIS
LIN {X 0.044,Y -378.879,Z 1226.620,A 0.000,B 0.000,C 90.000,E1 111.535} C_DIS
LIN {X 0.164,Y -393.852,Z 1226.607,A 0.000,B 0.000,C 90.000,E1 109.214} C_DIS
LIN {X 0.029,Y -410.296,Z 1226.594,A 0.000,B 0.000,C 90.000,E1 106.985} C_DIS
LIN {X 0.172,Y -428.329,Z 1226.582,A 0.000,B 0.000,C 90.000,E1 104.773} C_DIS
LIN {X -0.179,Y -447.903,Z 1226.570,A 0.000,B 0.000,C 90.000,E1 102.703} C_DIS
LIN {X 0.085,Y -468.187,Z 1226.560,A 0.000,B 0.000,C 90.000,E1 100.715} C_DIS
LIN {X 0.067,Y -473.221,Z 1226.557,A 0.000,B 0.000,C 90.000,E1 100.254} C_DIS
LIN {X 0.121,Y -475.107,Z 1226.556,A 0.000,B 0.000,C 90.000,E1 100.018} C_DIS
LIN {X -0.096,Y -476.679,Z 1226.554,A 0.000,B 0.000,C 90.000,E1 99.792} C_DIS
LIN {X -0.234,Y -477.857,Z 1226.553,A 0.000,B 0.000,C 90.000,E1 99.557} C_DIS
LIN {X -0.021,Y -479.281,Z 1226.550,A 0.000,B 0.000,C 90.000,E1 99.029} C_DIS
LIN {X 0.125,Y -479.669,Z 1226.547,A 0.000,B 0.000,C 90.000,E1 98.511} C_DIS
LIN {X -0.194,Y -479.087,Z 1226.545,A 0.000,B 0.000,C 90.000,E1 98.049} C_DIS
LIN {X -0.034,Y -477.442,Z 1226.542,A 0.000,B 0.000,C 90.000,E1 97.530} C_DIS
LIN {X -0.161,Y -476.131,Z 1226.540,A 0.000,B 0.000,C 90.000,E1 97.296} C_DIS
LIN {X -0.086,Y -466.944,Z 1226.533,A 0.000,B 0.000,C 90.000,E1 96.030} C_DIS
LIN {X 0.135,Y -449.134,Z 1226.519,A 0.000,B 0.000,C 90.000,E1 93.440} C_DIS
LIN {X -0.060,Y -430.619,Z 1226.503,A 0.000,B 0.000,C 90.000,E1 90.573} C_DIS
LIN {X 0.121,Y -412.668,Z 1226.485,A 0.000,B 0.000,C 90.000,E1 87.306} C_DIS
LIN {X -0.139,Y -402.624,Z 1226.474,A 0.000,B 0.000,C 90.000,E1 85.412} C_DIS
LIN {X -0.194,Y -393.944,Z 1226.465,A 0.000,B 0.000,C 90.000,E1 83.742} C_DIS
LIN {X 0.016,Y -383.718,Z 1226.454,A 0.000,B 0.000,C 90.000,E1 81.724} C_DIS
LIN {X 0.104,Y -374.765,Z 1226.444,A 0.000,B 0.000,C 90.000,E1 79.982} C_DIS
LIN {X 0.112,Y -367.068,Z 1226.436,A 0.000,B 0.000,C 90.000,E1 78.522} C_DIS
LIN {X 0.046,Y -357.602,Z 1226.427,A 0.000,B 0.000,C 90.000,E1 76.756} C_DIS
LIN {X 0.167,Y -346.347,Z 1226.415,A 0.000,B 0.000,C 90.000,E1 74.629} C_DIS
LIN {X 0.132,Y -335.091,Z 1226.403,A 0.000,B 0.000,C 90.000,E1 72.489} C_DIS
LIN {X 0.009,Y -322.480,Z 1226.389,A 0.000,B 0.000,C 90.000,E1 70.007} C_DIS
LIN {X -0.039,Y -306.167,Z 1226.369,A 0.000,B 0.000,C 90.000,E1 66.485} C_DIS
LIN {X 0.014,Y -292.574,Z 1226.351,A 0.000,B 0.000,C 90.000,E1 63.179} C_DIS
LIN {X 0.053,Y -280.003,Z 1226.332,A 0.000,B 0.000,C 90.000,E1 59.793} C_DIS
LIN {X 0.032,Y -268.443,Z 1226.313,A 0.000,B 0.000,C 90.000,E1 56.342} C_DIS
LIN {X -0.141,Y -258.829,Z 1226.295,A 0.000,B 0.000,C 90.000,E1 53.210} C_DIS
LIN {X 0.023,Y -248.933,Z 1226.276,A 0.000,B 0.000,C 90.000,E1 49.585} C_DIS
LIN {X 0.031,Y -241.506,Z 1226.259,A 0.000,B 0.000,C 90.000,E1 46.662} C_DIS
LIN {X 0.004,Y -234.406,Z 1226.243,A 0.000,B 0.000,C 90.000,E1 43.704} C_DIS
LIN {X -0.016,Y -227.500,Z 1226.226,A 0.000,B 0.000,C 90.000,E1 40.701} C_DIS
LIN {X 0.025,Y -219.400,Z 1226.205,A 0.000,B 0.000,C 90.000,E1 36.870} C_DIS
LIN {X -0.043,Y -213.513,Z 1226.188,A 0.000,B 0.000,C 90.000,E1 33.785} C_DIS
LIN {X -0.111,Y -207.025,Z 1226.166,A 0.000,B 0.000,C 90.000,E1 29.873} C_DIS
LIN {X 0.031,Y -201.554,Z 1226.144,A 0.000,B 0.000,C 90.000,E1 25.848} C_DIS
LIN {X -0.068,Y -196.964,Z 1226.121,A 0.000,B 0.000,C 90.000,E1 21.844} C_DIS
LIN {X -0.040,Y -193.235,Z 1226.099,A 0.000,B 0.000,C 90.000,E1 17.764} C_DIS
LIN {X -0.010,Y -189.862,Z 1226.071,A 0.000,B 0.000,C 90.000,E1 12.827} C_DIS
LIN {X 0.004,Y -187.359,Z 1226.034,A 0.000,B 0.000,C 90.000,E1 6.201} C_DIS
LIN {X 0.083,Y -188.651,Z 1225.974,A 0.000,B 0.000,C 90.000,E1 355.355} C_DIS
LIN {X 0.054,Y -191.890,Z 1225.942,A 0.000,B 0.000,C 90.000,E1 349.577} C_DIS
LIN {X -0.046,Y -196.014,Z 1225.915,A 0.000,B 0.000,C 90.000,E1 344.685} C_DIS
LIN {X 0.003,Y -200.347,Z 1225.892,A 0.000,B 0.000,C 90.000,E1 340.604} C_DIS
LIN {X -0.120,Y -205.517,Z 1225.870,A 0.000,B 0.000,C 90.000,E1 336.613} C_DIS
LIN {X -0.054,Y -211.298,Z 1225.848,A 0.000,B 0.000,C 90.000,E1 332.615} C_DIS
LIN {X 0.032,Y -217.545,Z 1225.826,A 0.000,B 0.000,C 90.000,E1 328.663} C_DIS
LIN {X 0.104,Y -224.468,Z 1225.804,A 0.000,B 0.000,C 90.000,E1 324.769} C_DIS
LIN {X 0.046,Y -232.030,Z 1225.783,A 0.000,B 0.000,C 90.000,E1 320.964} C_DIS
LIN {X -0.049,Y -240.498,Z 1225.762,A 0.000,B 0.000,C 90.000,E1 317.229} C_DIS
LIN {X 0.131,Y -247.145,Z 1225.748,A 0.000,B 0.000,C 90.000,E1 314.595} C_DIS
LIN {X 0.154,Y -255.852,Z 1225.732,A 0.000,B 0.000,C 90.000,E1 311.676} C_DIS
LIN {X 0.028,Y -264.657,Z 1225.718,A 0.000,B 0.000,C 90.000,E1 309.197} C_DIS
LIN {X -0.022,Y -274.444,Z 1225.704,A 0.000,B 0.000,C 90.000,E1 306.744} C_DIS
LIN {X -0.059,Y -287.113,Z 1225.689,A 0.000,B 0.000,C 90.000,E1 303.992} C_DIS
LIN {X 0.162,Y -303.118,Z 1225.672,A 0.000,B 0.000,C 90.000,E1 300.924} C_DIS
LIN {X -0.181,Y -308.893,Z 1225.667,A 0.000,B 0.000,C 90.000,E1 300.001} C_DIS
LIN {X -0.061,Y -315.419,Z 1225.661,A 0.000,B 0.000,C 90.000,E1 298.999} C_DIS
LIN {X -0.075,Y -330.179,Z 1225.650,A 0.000,B 0.000,C 90.000,E1 297.078} C_DIS
LIN {X -0.024,Y -348.654,Z 1225.638,A 0.000,B 0.000,C 90.000,E1 294.899} C_DIS
LIN {X -0.026,Y -372.474,Z 1225.624,A 0.000,B 0.000,C 90.000,E1 292.280} C_DIS
LIN {X -0.106,Y -385.514,Z 1225.616,A 0.000,B 0.000,C 90.000,E1 290.918} C_DIS
LIN {X 0.076,Y -401.021,Z 1225.607,A 0.000,B 0.000,C 90.000,E1 289.268} C_DIS
LIN {X 0.077,Y -413.884,Z 1225.600,A 0.000,B 0.000,C 90.000,E1 287.946} C_DIS
LIN {X -0.051,Y -421.462,Z 1225.595,A 0.000,B 0.000,C 90.000,E1 287.166} C_DIS
LIN {X 0.254,Y -428.708,Z 1225.591,A 0.000,B 0.000,C 90.000,E1 286.315} C_DIS
LIN {X -0.069,Y -435.474,Z 1225.586,A 0.000,B 0.000,C 90.000,E1 285.552} C_DIS
LIN {X 0.202,Y -441.625,Z 1225.582,A 0.000,B 0.000,C 90.000,E1 284.717} C_DIS
LIN {X -0.006,Y -447.135,Z 1225.578,A 0.000,B 0.000,C 90.000,E1 283.953} C_DIS
LIN {X -0.066,Y -452.041,Z 1225.573,A 0.000,B 0.000,C 90.000,E1 283.175} C_DIS
LIN {X -0.189,Y -456.276,Z 1225.569,A 0.000,B 0.000,C 90.000,E1 282.411} C_DIS
LIN {X 0.169,Y -459.813,Z 1225.564,A 0.000,B 0.000,C 90.000,E1 281.591} C_DIS
LIN {X 0.190,Y -461.797,Z 1225.562,A 0.000,B 0.000,C 90.000,E1 281.074} C_DIS
LIN {X -0.147,Y -463.537,Z 1225.559,A 0.000,B 0.000,C 90.000,E1 280.602} C_DIS
LIN {X -0.021,Y -464.996,Z 1225.556,A 0.000,B 0.000,C 90.000,E1 280.074} C_DIS
LIN {X 0.035,Y -466.208,Z 1225.553,A 0.000,B 0.000,C 90.000,E1 279.557} C_DIS
LIN {X 0.177,Y -467.134,Z 1225.550,A 0.000,B 0.000,C 90.000,E1 279.029} C_DIS
LIN {X -0.209,Y -467.818,Z 1225.547,A 0.000,B 0.000,C 90.000,E1 278.568} C_DIS
LIN {X -0.126,Y -468.191,Z 1225.545,A 0.000,B 0.000,C 90.000,E1 278.049} C_DIS
LIN {X -0.037,Y -468.214,Z 1225.542,A 0.000,B 0.000,C 90.000,E1 277.530} C_DIS
LIN {X 0.113,Y -467.887,Z 1225.539,A 0.000,B 0.000,C 90.000,E1 277.004} C_DIS
LIN {X 0.202,Y -467.135,Z 1225.536,A 0.000,B 0.000,C 90.000,E1 276.486} C_DIS
LIN {X -0.173,Y -465.950,Z 1225.533,A 0.000,B 0.000,C 90.000,E1 276.024} C_DIS
LIN {X -0.135,Y -464.369,Z 1225.531,A 0.000,B 0.000,C 90.000,E1 275.511} C_DIS
LIN {X -0.057,Y -462.346,Z 1225.528,A 0.000,B 0.000,C 90.000,E1 274.992} C_DIS
LIN {X 0.012,Y -459.859,Z 1225.525,A 0.000,B 0.000,C 90.000,E1 274.473} C_DIS
LIN {X 0.057,Y -456.696,Z 1225.522,A 0.000,B 0.000,C 90.000,E1 273.955} C_DIS
LIN {X 0.056,Y -452.735,Z 1225.519,A 0.000,B 0.000,C 90.000,E1 273.440} C_DIS
LIN {X -0.178,Y -450.369,Z 1225.518,A 0.000,B 0.000,C 90.000,E1 273.212} C_DIS
LIN {X 0.062,Y -447.687,Z 1225.516,A 0.000,B 0.000,C 90.000,E1 272.922} C_DIS
LIN {X -0.071,Y -444.819,Z 1225.515,A 0.000,B 0.000,C 90.000,E1 272.694} C_DIS
LIN {X -0.057,Y -438.534,Z 1225.512,A 0.000,B 0.000,C 90.000,E1 272.236} C_DIS
LIN {X 0.079,Y -431.771,Z 1225.510,A 0.000,B 0.000,C 90.000,E1 271.835} C_DIS
LIN {X -0.116,Y -424.694,Z 1225.509,A 0.000,B 0.000,C 90.000,E1 271.547} C_DIS
LIN {X 0.075,Y -417.762,Z 1225.507,A 0.000,B 0.000,C 90.000,E1 271.260} C_DIS
LIN {X 0.138,Y -410.850,Z 1225.506,A 0.000,B 0.000,C 90.000,E1 271.031} C_DIS
LIN {X -0.190,Y -400.159,Z 1225.504,A 0.000,B 0.000,C 90.000,E1 270.802} C_DIS
LIN {X -0.063,Y -393.162,Z 1225.503,A 0.000,B 0.000,C 90.000,E1 270.630} C_DIS
LIN {X -0.186,Y -384.905,Z 1225.503,A 0.000,B 0.000,C 90.000,E1 270.516} C_DIS
LIN {X -0.106,Y -374.503,Z 1225.502,A 0.000,B 0.000,C 90.000,E1 270.401} C_DIS
LIN {X -0.041,Y -365.626,Z 1225.502,A 0.000,B 0.000,C 90.000,E1 270.344} C_DIS
LIN {X -0.050,Y -181.580,Z 1225.502,A 0.000,B 0.000,C 90.000,E1 270.344} C_DIS
LIN {X 0.083,Y -180.842,Z 1225.472,A 0.000,B 0.000,C 90.000,E1 264.894} C_DIS
LIN {X -0.014,Y -178.950,Z 1225.444,A 0.000,B 0.000,C 90.000,E1 259.859} C_DIS
LIN {X 0.003,Y -176.855,Z 1225.425,A 0.000,B 0.000,C 90.000,E1 256.464} C_DIS
LIN {X -0.026,Y -175.514,Z 1225.411,A 0.000,B 0.000,C 90.000,E1 253.921} C_DIS
LIN {X -0.024,Y -172.253,Z 1225.387,A 0.000,B 0.000,C 90.000,E1 249.645} C_DIS
LIN {X 0.015,Y -171.732,Z 1225.382,A 0.000,B 0.000,C 90.000,E1 248.773} C_DIS
LIN {X 0.024,Y -167.328,Z 1225.353,A 0.000,B 0.000,C 90.000,E1 243.589} C_DIS
LIN {X -0.044,Y -166.712,Z 1225.349,A 0.000,B 0.000,C 90.000,E1 242.743} C_DIS
LIN {X 0.094,Y -162.692,Z 1225.324,A 0.000,B 0.000,C 90.000,E1 238.329} C_DIS
LIN {X -0.068,Y -161.383,Z 1225.314,A 0.000,B 0.000,C 90.000,E1 236.628} C_DIS
LIN {X -0.025,Y -157.376,Z 1225.290,A 0.000,B 0.000,C 90.000,E1 232.190} C_DIS
LIN {X 0.009,Y -155.369,Z 1225.275,A 0.000,B 0.000,C 90.000,E1 229.504} C_DIS
LIN {X 0.056,Y -151.709,Z 1225.250,A 0.000,B 0.000,C 90.000,E1 225.000} C_DIS
LIN {X 0.066,Y -149.901,Z 1225.235,A 0.000,B 0.000,C 90.000,E1 222.285} C_DIS
LIN {X 0.089,Y -146.759,Z 1225.210,A 0.000,B 0.000,C 90.000,E1 217.729} C_DIS
LIN {X -0.013,Y -145.327,Z 1225.195,A 0.000,B 0.000,C 90.000,E1 215.025} C_DIS
LIN {X 0.028,Y -142.410,Z 1225.164,A 0.000,B 0.000,C 90.000,E1 209.489} C_DIS
LIN {X -0.047,Y -141.394,Z 1225.148,A 0.000,B 0.000,C 90.000,E1 206.744} C_DIS
LIN {X -0.058,Y -139.353,Z 1225.112,A 0.000,B 0.000,C 90.000,E1 200.248} C_DIS
LIN {X 0.062,Y -138.792,Z 1225.097,A 0.000,B 0.000,C 90.000,E1 197.402} C_DIS
LIN {X -0.016,Y -138.346,Z 1225.055,A 0.000,B 0.000,C 90.000,E1 189.962} C_DIS
LIN {X 0.001,Y -139.379,Z 1225.009,A 0.000,B 0.000,C 90.000,E1 181.547} C_DIS
LIN {X 0.055,Y -141.271,Z 1224.972,A 0.000,B 0.000,C 90.000,E1 175.008} C_DIS
LIN {X 0.013,Y -142.637,Z 1224.957,A 0.000,B 0.000,C 90.000,E1 172.243} C_DIS
LIN {X -0.035,Y -144.966,Z 1224.931,A 0.000,B 0.000,C 90.000,E1 167.645} C_DIS
LIN {X -0.045,Y -147.594,Z 1224.911,A 0.000,B 0.000,C 90.000,E1 163.976} C_DIS
LIN {X -0.015,Y -150.211,Z 1224.891,A 0.000,B 0.000,C 90.000,E1 160.315} C_DIS
LIN {X 0.052,Y -153.597,Z 1224.870,A 0.000,B 0.000,C 90.000,E1 156.666} C_DIS
LIN {X 0.040,Y -157.013,Z 1224.850,A 0.000,B 0.000,C 90.000,E1 153.076} C_DIS
LIN {X -0.027,Y -161.133,Z 1224.831,A 0.000,B 0.000,C 90.000,E1 149.537} C_DIS
LIN {X -0.082,Y -163.232,Z 1224.821,A 0.000,B 0.000,C 90.000,E1 147.788} C_DIS
LIN {X -0.079,Y -167.665,Z 1224.801,A 0.000,B 0.000,C 90.000,E1 144.276} C_DIS
LIN {X 0.069,Y -171.488,Z 1224.787,A 0.000,B 0.000,C 90.000,E1 141.618} C_DIS
LIN {X 0.114,Y -176.419,Z 1224.768,A 0.000,B 0.000,C 90.000,E1 138.162} C_DIS
LIN {X -0.015,Y -180.715,Z 1224.754,A 0.000,B 0.000,C 90.000,E1 135.648} C_DIS
LIN {X -0.034,Y -186.118,Z 1224.735,A 0.000,B 0.000,C 90.000,E1 132.285} C_DIS
LIN {X 0.024,Y -190.755,Z 1224.721,A 0.000,B 0.000,C 90.000,E1 129.769} C_DIS
LIN {X -0.067,Y -196.510,Z 1224.703,A 0.000,B 0.000,C 90.000,E1 126.503} C_DIS
LIN {X -0.020,Y -201.032,Z 1224.690,A 0.000,B 0.000,C 90.000,E1 124.199} C_DIS
LIN {X -0.067,Y -310.786,Z 1224.690,A 0.000,B 0.000,C 90.000,E1 124.199} C_DIS
LIN {X -0.173,Y -312.265,Z 1224.690,A 0.000,B 0.000,C 90.000,E1 124.199} C_DIS
LIN {X 0.016,Y -315.723,Z 1224.689,A 0.000,B 0.000,C 90.000,E1 124.040} C_DIS
LIN {X -0.091,Y -318.967,Z 1224.688,A 0.000,B 0.000,C 90.000,E1 123.833} C_DIS
LIN {X 0.164,Y -322.645,Z 1224.686,A 0.000,B 0.000,C 90.000,E1 123.372} C_DIS
LIN {X 0.053,Y -324.533,Z 1224.684,A 0.000,B 0.000,C 90.000,E1 123.086} C_DIS
LIN {X -0.059,Y -326.010,Z 1224.682,A 0.000,B 0.000,C 90.000,E1 122.801} C_DIS
LIN {X 0.034,Y -339.293,Z 1224.663,A 0.000,B 0.000,C 90.000,E1 119.333} C_DIS
LIN {X 0.049,Y -351.613,Z 1224.648,A 0.000,B 0.000,C 90.000,E1 116.565} C_DIS
LIN {X -0.207,Y -365.420,Z 1224.633,A 0.000,B 0.000,C 90.000,E1 113.898} C_DIS
LIN {X -0.158,Y -379.042,Z 1224.620,A 0.000,B 0.000,C 90.000,E1 111.535} C_DIS
LIN {X -0.042,Y -394.033,Z 1224.607,A 0.000,B 0.000,C 90.000,E1 109.214} C_DIS
LIN {X -0.061,Y -410.498,Z 1224.594,A 0.000,B 0.000,C 90.000,E1 106.968} C_DIS
LIN {X -0.042,Y -428.552,Z 1224.582,A 0.000,B 0.000,C 90.000,E1 104.773} C_DIS
LIN {X 0.047,Y -448.138,Z 1224.570,A 0.000,B 0.000,C 90.000,E1 102.647} C_DIS
LIN {X -0.118,Y -468.430,Z 1224.559,A 0.000,B 0.000,C 90.000,E1 100.715} C_DIS
LIN {X -0.134,Y -473.400,Z 1224.557,A 0.000,B 0.000,C 90.000,E1 100.254} C_DIS
LIN {X -0.079,Y -475.211,Z 1224.556,A 0.000,B 0.000,C 90.000,E1 100.018} C_DIS
LIN {X 0.253,Y -476.726,Z 1224.554,A 0.000,B 0.000,C 90.000,E1 99.726} C_DIS
LIN {X 0.037,Y -477.858,Z 1224.553,A 0.000,B 0.000,C 90.000,E1 99.500} C_DIS
LIN {X 0.251,Y -479.209,Z 1224.550,A 0.000,B 0.000,C 90.000,E1 98.973} C_DIS
LIN {X -0.076,Y -479.535,Z 1224.547,A 0.000,B 0.000,C 90.000,E1 98.511} C_DIS
LIN {X 0.080,Y -478.890,Z 1224.544,A 0.000,B 0.000,C 90.000,E1 97.992} C_DIS
LIN {X -0.235,Y -477.169,Z 1224.542,A 0.000,B 0.000,C 90.000,E1 97.530} C_DIS
LIN {X 0.110,Y -475.810,Z 1224.540,A 0.000,B 0.000,C 90.000,E1 97.239} C_DIS
LIN {X -0.119,Y -459.370,Z 1224.528,A 0.000,B 0.000,C 90.000,E1 94.992} C_DIS
LIN {X -0.086,Y -445.312,Z 1224.516,A 0.000,B 0.000,C 90.000,E1 92.922} C_DIS
LIN {X -0.116,Y -428.724,Z 1224.501,A 0.000,B 0.000,C 90.000,E1 90.286} C_DIS
LIN {X -0.087,Y -412.368,Z 1224.485,A 0.000,B 0.000,C 90.000,E1 87.306} C_DIS
LIN {X 0.053,Y -402.308,Z 1224.474,A 0.000,B 0.000,C 90.000,E1 85.355} C_DIS
LIN {X -0.012,Y -393.621,Z 1224.465,A 0.000,B 0.000,C 90.000,E1 83.685} C_DIS
LIN {X -0.194,Y -383.394,Z 1224.454,A 0.000,B 0.000,C 90.000,E1 81.724} C_DIS
LIN {X -0.108,Y -374.451,Z 1224.444,A 0.000,B 0.000,C 90.000,E1 79.982} C_DIS
LIN {X -0.115,Y -365.180,Z 1224.434,A 0.000,B 0.000,C 90.000,E1 78.229} C_DIS
LIN {X 0.137,Y -355.649,Z 1224.425,A 0.000,B 0.000,C 90.000,E1 76.408} C_DIS
LIN {X -0.120,Y -344.424,Z 1224.413,A 0.000,B 0.000,C 90.000,E1 74.338} C_DIS
LIN {X -0.111,Y -331.603,Z 1224.399,A 0.000,B 0.000,C 90.000,E1 71.873} C_DIS
LIN {X -0.060,Y -317.600,Z 1224.383,A 0.000,B 0.000,C 90.000,E1 69.028} C_DIS
LIN {X -0.141,Y -301.704,Z 1224.364,A 0.000,B 0.000,C 90.000,E1 65.485} C_DIS
LIN {X -0.091,Y -288.449,Z 1224.345,A 0.000,B 0.000,C 90.000,E1 62.153} C_DIS
LIN {X -0.043,Y -276.139,Z 1224.326,A 0.000,B 0.000,C 90.000,E1 58.742} C_DIS
LIN {X -0.042,Y -264.855,Z 1224.307,A 0.000,B 0.000,C 90.000,E1 55.261} C_DIS
LIN {X 0.025,Y -254.446,Z 1224.287,A 0.000,B 0.000,C 90.000,E1 51.698} C_DIS
LIN {X 0.014,Y -244.808,Z 1224.267,A 0.000,B 0.000,C 90.000,E1 48.081} C_DIS
LIN {X 0.013,Y -235.738,Z 1224.247,A 0.000,B 0.000,C 90.000,E1 44.393} C_DIS
LIN {X 0.021,Y -228.781,Z 1224.230,A 0.000,B 0.000,C 90.000,E1 41.391} C_DIS
LIN {X -0.069,Y -220.494,Z 1224.209,A 0.000,B 0.000,C 90.000,E1 37.604} C_DIS
LIN {X 0.015,Y -213.041,Z 1224.187,A 0.000,B 0.000,C 90.000,E1 33.706} C_DIS
LIN {X -0.074,Y -206.594,Z 1224.165,A 0.000,B 0.000,C 90.000,E1 29.795} C_DIS
LIN {X -0.040,Y -201.174,Z 1224.143,A 0.000,B 0.000,C 90.000,E1 25.796} C_DIS
LIN {X -0.070,Y -196.604,Z 1224.121,A 0.000,B 0.000,C 90.000,E1 21.770} C_DIS
LIN {X -0.062,Y -192.860,Z 1224.098,A 0.000,B 0.000,C 90.000,E1 17.692} C_DIS
LIN {X -0.098,Y -189.510,Z 1224.071,A 0.000,B 0.000,C 90.000,E1 12.771} C_DIS
LIN {X -0.095,Y -187.023,Z 1224.034,A 0.000,B 0.000,C 90.000,E1 6.144} C_DIS
LIN {X 0.072,Y -188.334,Z 1223.974,A 0.000,B 0.000,C 90.000,E1 355.355} C_DIS
LIN {X 0.030,Y -191.568,Z 1223.942,A 0.000,B 0.000,C 90.000,E1 349.577} C_DIS
LIN {X 0.106,Y -195.722,Z 1223.915,A 0.000,B 0.000,C 90.000,E1 344.629} C_DIS
LIN {X -0.043,Y -200.087,Z 1223.892,A 0.000,B 0.000,C 90.000,E1 340.604} C_DIS
LIN {X 0.013,Y -205.278,Z 1223.870,A 0.000,B 0.000,C 90.000,E1 336.561} C_DIS
LIN {X -0.118,Y -211.091,Z 1223.848,A 0.000,B 0.000,C 90.000,E1 332.615} C_DIS
LIN {X 0.093,Y -216.072,Z 1223.830,A 0.000,B 0.000,C 90.000,E1 329.410} C_DIS
LIN {X -0.008,Y -222.837,Z 1223.809,A 0.000,B 0.000,C 90.000,E1 325.548} C_DIS
LIN {X 0.060,Y -230.293,Z 1223.787,A 0.000,B 0.000,C 90.000,E1 321.698} C_DIS
LIN {X 0.089,Y -238.574,Z 1223.766,A 0.000,B 0.000,C 90.000,E1 317.919} C_DIS
LIN {X 0.026,Y -247.031,Z 1223.748,A 0.000,B 0.000,C 90.000,E1 314.595} C_DIS
LIN {X 0.019,Y -254.628,Z 1223.734,A 0.000,B 0.000,C 90.000,E1 312.043} C_DIS
LIN {X -0.137,Y -263.314,Z 1223.720,A 0.000,B 0.000,C 90.000,E1 309.564} C_DIS
LIN {X -0.065,Y -272.960,Z 1223.706,A 0.000,B 0.000,C 90.000,E1 307.076} C_DIS
LIN {X 0.087,Y -285.455,Z 1223.691,A 0.000,B 0.000,C 90.000,E1 304.278} C_DIS
LIN {X 0.010,Y -299.416,Z 1223.676,A 0.000,B 0.000,C 90.000,E1 301.592} C_DIS
LIN {X 0.103,Y -308.807,Z 1223.666,A 0.000,B 0.000,C 90.000,E1 299.922} C_DIS
LIN {X 0.074,Y -315.315,Z 1223.661,A 0.000,B 0.000,C 90.000,E1 298.949} C_DIS
LIN {X -0.075,Y -330.110,Z 1223.650,A 0.000,B 0.000,C 90.000,E1 297.052} C_DIS
LIN {X -0.056,Y -348.418,Z 1223.638,A 0.000,B 0.000,C 90.000,E1 294.899} C_DIS
LIN {X 0.111,Y -372.029,Z 1223.624,A 0.000,B 0.000,C 90.000,E1 292.280} C_DIS
LIN {X 0.051,Y -385.114,Z 1223.616,A 0.000,B 0.000,C 90.000,E1 290.918} C_DIS
LIN {X 0.189,Y -400.757,Z 1223.607,A 0.000,B 0.000,C 90.000,E1 289.268} C_DIS
LIN {X 0.149,Y -413.712,Z 1223.600,A 0.000,B 0.000,C 90.000,E1 287.946} C_DIS
LIN {X -0.092,Y -423.771,Z 1223.594,A 0.000,B 0.000,C 90.000,E1 286.913} C_DIS
LIN {X 0.093,Y -430.871,Z 1223.589,A 0.000,B 0.000,C 90.000,E1 286.079} C_DIS
LIN {X -0.103,Y -437.451,Z 1223.585,A 0.000,B 0.000,C 90.000,E1 285.300} C_DIS
LIN {X 0.075,Y -443.403,Z 1223.580,A 0.000,B 0.000,C 90.000,E1 284.481} C_DIS
LIN {X -0.017,Y -448.746,Z 1223.576,A 0.000,B 0.000,C 90.000,E1 283.703} C_DIS
LIN {X -0.168,Y -453.500,Z 1223.572,A 0.000,B 0.000,C 90.000,E1 282.939} C_DIS
LIN {X 0.164,Y -457.498,Z 1223.567,A 0.000,B 0.000,C 90.000,E1 282.119} C_DIS
LIN {X 0.167,Y -459.809,Z 1223.565,A 0.000,B 0.000,C 90.000,E1 281.602} C_DIS
LIN {X -0.172,Y -461.817,Z 1223.562,A 0.000,B 0.000,C 90.000,E1 281.130} C_DIS
LIN {X -0.056,Y -463.571,Z 1223.559,A 0.000,B 0.000,C 90.000,E1 280.602} C_DIS
LIN {X 0.071,Y -465.079,Z 1223.556,A 0.000,B 0.000,C 90.000,E1 280.074} C_DIS
LIN {X 0.127,Y -466.284,Z 1223.553,A 0.000,B 0.000,C 90.000,E1 279.557} C_DIS
LIN {X -0.191,Y -467.201,Z 1223.550,A 0.000,B 0.000,C 90.000,E1 279.086} C_DIS
LIN {X -0.116,Y -467.900,Z 1223.547,A 0.000,B 0.000,C 90.000,E1 278.568} C_DIS
LIN {X -0.033,Y -468.276,Z 1223.545,A 0.000,B 0.000,C 90.000,E1 278.049} C_DIS
LIN {X 0.057,Y -468.343,Z 1223.542,A 0.000,B 0.000,C 90.000,E1 277.530} C_DIS
LIN {X 0.150,Y -468.000,Z 1223.539,A 0.000,B 0.000,C 90.000,E1 277.011} C_DIS
LIN {X -0.167,Y -467.297,Z 1223.536,A 0.000,B 0.000,C 90.000,E1 276.543} C_DIS
LIN {X -0.127,Y -466.155,Z 1223.533,A 0.000,B 0.000,C 90.000,E1 276.030} C_DIS
LIN {X -0.039,Y -464.609,Z 1223.531,A 0.000,B 0.000,C 90.000,E1 275.511} C_DIS
LIN {X 0.040,Y -462.649,Z 1223.528,A 0.000,B 0.000,C 90.000,E1 274.992} C_DIS
LIN {X 0.109,Y -460.188,Z 1223.525,A 0.000,B 0.000,C 90.000,E1 274.473} C_DIS
LIN {X 0.156,Y -457.072,Z 1223.522,A 0.000,B 0.000,C 90.000,E1 273.955} C_DIS
LIN {X 0.156,Y -453.136,Z 1223.519,A 0.000,B 0.000,C 90.000,E1 273.440} C_DIS
LIN {X -0.078,Y -450.799,Z 1223.518,A 0.000,B 0.000,C 90.000,E1 273.212} C_DIS
LIN {X 0.163,Y -448.157,Z 1223.516,A 0.000,B 0.000,C 90.000,E1 272.922} C_DIS
LIN {X -0.138,Y -442.138,Z 1223.514,A 0.000,B 0.000,C 90.000,E1 272.465} C_DIS
LIN {X 0.080,Y -435.398,Z 1223.511,A 0.000,B 0.000,C 90.000,E1 272.007} C_DIS
LIN {X 0.000,Y -428.211,Z 1223.509,A 0.000,B 0.000,C 90.000,E1 271.661} C_DIS
LIN {X 0.015,Y -417.886,Z 1223.507,A 0.000,B 0.000,C 90.000,E1 271.260} C_DIS
LIN {X 0.101,Y -411.140,Z 1223.506,A 0.000,B 0.000,C 90.000,E1 271.031} C_DIS
LIN {X 0.190,Y -400.665,Z 1223.504,A 0.000,B 0.000,C 90.000,E1 270.745} C_DIS
LIN {X -0.098,Y -393.694,Z 1223.503,A 0.000,B 0.000,C 90.000,E1 270.630} C_DIS
LIN {X 0.144,Y -385.388,Z 1223.503,A 0.000,B 0.000,C 90.000,E1 270.458} C_DIS
LIN {X -0.168,Y -375.291,Z 1223.502,A 0.000,B 0.000,C 90.000,E1 270.401} C_DIS
LIN {X -0.168,Y -364.059,Z 1223.502,A 0.000,B 0.000,C 90.000,E1 270.344} C_DIS
LIN {X 0.067,Y -181.581,Z 1223.502,A 0.000,B 0.000,C 90.000,E1 270.286} C_DIS
LIN {X 0.048,Y -180.838,Z 1223.472,A 0.000,B 0.000,C 90.000,E1 264.894} C_DIS
LIN {X -0.049,Y -178.946,Z 1223.444,A 0.000,B 0.000,C 90.000,E1 259.859} C_DIS
LIN {X 0.046,Y -176.401,Z 1223.420,A 0.000,B 0.000,C 90.000,E1 255.589} C_DIS
LIN {X -0.060,Y -175.506,Z 1223.411,A 0.000,B 0.000,C 90.000,E1 253.921} C_DIS
LIN {X 0.002,Y -172.246,Z 1223.387,A 0.000,B 0.000,C 90.000,E1 249.625} C_DIS
LIN {X -0.019,Y -171.724,Z 1223.382,A 0.000,B 0.000,C 90.000,E1 248.773} C_DIS
LIN {X -0.010,Y -167.321,Z 1223.353,A 0.000,B 0.000,C 90.000,E1 243.589} C_DIS
LIN {X -0.077,Y -166.703,Z 1223.348,A 0.000,B 0.000,C 90.000,E1 242.743} C_DIS
LIN {X 0.061,Y -162.684,Z 1223.324,A 0.000,B 0.000,C 90.000,E1 238.329} C_DIS
LIN {X 0.034,Y -161.374,Z 1223.314,A 0.000,B 0.000,C 90.000,E1 236.580} C_DIS
LIN {X -0.057,Y -157.367,Z 1223.290,A 0.000,B 0.000,C 90.000,E1 232.190} C_DIS
LIN {X 0.095,Y -155.358,Z 1223.275,A 0.000,B 0.000,C 90.000,E1 229.461} C_DIS
LIN {X 0.024,Y -151.701,Z 1223.250,A 0.000,B 0.000,C 90.000,E1 225.000} C_DIS
LIN {X -0.038,Y -150.562,Z 1223.240,A 0.000,B 0.000,C 90.000,E1 223.218} C_DIS
LIN {X -0.011,Y -147.289,Z 1223.215,A 0.000,B 0.000,C 90.000,E1 218.669} C_DIS
LIN {X -0.043,Y -145.319,Z 1223.194,A 0.000,B 0.000,C 90.000,E1 215.025} C_DIS
LIN {X -0.003,Y -142.405,Z 1223.164,A 0.000,B 0.000,C 90.000,E1 209.489} C_DIS
LIN {X -0.076,Y -141.388,Z 1223.148,A 0.000,B 0.000,C 90.000,E1 206.744} C_DIS
LIN {X 0.042,Y -139.351,Z 1223.112,A 0.000,B 0.000,C 90.000,E1 200.194} C_DIS
LIN {X 0.032,Y -138.790,Z 1223.097,A 0.000,B 0.000,C 90.000,E1 197.402} C_DIS
LIN {X -0.046,Y -138.346,Z 1223.055,A 0.000,B 0.000,C 90.000,E1 189.962} C_DIS
LIN {X -0.028,Y -139.382,Z 1223.009,A 0.000,B 0.000,C 90.000,E1 181.547} C_DIS
LIN {X 0.025,Y -141.277,Z 1222.972,A 0.000,B 0.000,C 90.000,E1 175.008} C_DIS
LIN {X -0.016,Y -142.642,Z 1222.957,A 0.000,B 0.000,C 90.000,E1 172.243} C_DIS
LIN {X -0.066,Y -144.974,Z 1222.931,A 0.000,B 0.000,C 90.000,E1 167.645} C_DIS
LIN {X 0.066,Y -147.601,Z 1222.911,A 0.000,B 0.000,C 90.000,E1 163.921} C_DIS
LIN {X 0.004,Y -150.221,Z 1222.891,A 0.000,B 0.000,C 90.000,E1 160.296} C_DIS
LIN {X 0.020,Y -153.610,Z 1222.870,A 0.000,B 0.000,C 90.000,E1 156.666} C_DIS
LIN {X 0.008,Y -157.025,Z 1222.850,A 0.000,B 0.000,C 90.000,E1 153.076} C_DIS
LIN {X -0.060,Y -161.147,Z 1222.831,A 0.000,B 0.000,C 90.000,E1 149.537} C_DIS
LIN {X 0.022,Y -163.245,Z 1222.821,A 0.000,B 0.000,C 90.000,E1 147.740} C_DIS
LIN {X -0.015,Y -167.681,Z 1222.801,A 0.000,B 0.000,C 90.000,E1 144.242} C_DIS
LIN {X 0.035,Y -171.503,Z 1222.787,A 0.000,B 0.000,C 90.000,E1 141.618} C_DIS
LIN {X 0.079,Y -176.437,Z 1222.768,A 0.000,B 0.000,C 90.000,E1 138.162} C_DIS
LIN {X -0.050,Y -180.733,Z 1222.754,A 0.000,B 0.000,C 90.000,E1 135.648} C_DIS
LIN {X -0.069,Y -186.137,Z 1222.735,A 0.000,B 0.000,C 90.000,E1 132.285} C_DIS
LIN {X -0.012,Y -190.775,Z 1222.721,A 0.000,B 0.000,C 90.000,E1 129.769} C_DIS
LIN {X 0.054,Y -196.531,Z 1222.703,A 0.000,B 0.000,C 90.000,E1 126.457} C_DIS
LIN {X -0.106,Y -201.073,Z 1222.690,A 0.000,B 0.000,C 90.000,E1 124.199} C_DIS
LIN {X -0.199,Y -310.534,Z 1222.690,A 0.000,B 0.000,C 90.000,E1 124.199} C_DIS
LIN {X -0.042,Y -315.494,Z 1222.689,A 0.000,B 0.000,C 90.000,E1 124.040} C_DIS
LIN {X 0.041,Y -318.448,Z 1222.688,A 0.000,B 0.000,C 90.000,E1 123.833} C_DIS
LIN {X -0.007,Y -322.169,Z 1222.686,A 0.000,B 0.000,C 90.000,E1 123.452} C_DIS
LIN {X -0.027,Y -324.091,Z 1222.684,A 0.000,B 0.000,C 90.000,E1 123.166} C_DIS
LIN {X -0.047,Y -325.602,Z 1222.683,A 0.000,B 0.000,C 90.000,E1 122.880} C_DIS
LIN {X 0.147,Y -328.045,Z 1222.679,A 0.000,B 0.000,C 90.000,E1 122.212} C_DIS
LIN {X 0.040,Y -338.942,Z 1222.663,A 0.000,B 0.000,C 90.000,E1 119.411} C_DIS
LIN {X -0.103,Y -351.221,Z 1222.648,A 0.000,B 0.000,C 90.000,E1 116.668} C_DIS
LIN {X -0.057,Y -364.984,Z 1222.633,A 0.000,B 0.000,C 90.000,E1 113.951} C_DIS
LIN {X -0.022,Y -378.565,Z 1222.620,A 0.000,B 0.000,C 90.000,E1 111.589} C_DIS
LIN {X 0.083,Y -393.511,Z 1222.607,A 0.000,B 0.000,C 90.000,E1 109.268} C_DIS
LIN {X -0.070,Y -409.926,Z 1222.595,A 0.000,B 0.000,C 90.000,E1 107.040} C_DIS
LIN {X 0.056,Y -427.928,Z 1222.582,A 0.000,B 0.000,C 90.000,E1 104.828} C_DIS
LIN {X 0.013,Y -447.481,Z 1222.571,A 0.000,B 0.000,C 90.000,E1 102.715} C_DIS
LIN {X -0.184,Y -467.756,Z 1222.560,A 0.000,B 0.000,C 90.000,E1 100.782} C_DIS
LIN {X -0.124,Y -472.816,Z 1222.557,A 0.000,B 0.000,C 90.000,E1 100.310} C_DIS
LIN {X -0.075,Y -474.742,Z 1222.556,A 0.000,B 0.000,C 90.000,E1 100.074} C_DIS
LIN {X 0.175,Y -476.342,Z 1222.555,A 0.000,B 0.000,C 90.000,E1 99.792} C_DIS
LIN {X 0.037,Y -477.542,Z 1222.553,A 0.000,B 0.000,C 90.000,E1 99.557} C_DIS
LIN {X 0.250,Y -479.002,Z 1222.550,A 0.000,B 0.000,C 90.000,E1 99.029} C_DIS
LIN {X -0.081,Y -479.422,Z 1222.547,A 0.000,B 0.000,C 90.000,E1 98.568} C_DIS
LIN {X 0.073,Y -478.872,Z 1222.545,A 0.000,B 0.000,C 90.000,E1 98.049} C_DIS
LIN {X -0.243,Y -477.265,Z 1222.542,A 0.000,B 0.000,C 90.000,E1 97.587} C_DIS
LIN {X 0.101,Y -475.979,Z 1222.541,A 0.000,B 0.000,C 90.000,E1 97.296} C_DIS
LIN {X 0.053,Y -470.510,Z 1222.536,A 0.000,B 0.000,C 90.000,E1 96.549} C_DIS
LIN {X 0.150,Y -454.252,Z 1222.524,A 0.000,B 0.000,C 90.000,E1 94.245} C_DIS
LIN {X -0.036,Y -437.038,Z 1222.509,A 0.000,B 0.000,C 90.000,E1 91.661} C_DIS
LIN {X 0.167,Y -425.844,Z 1222.499,A 0.000,B 0.000,C 90.000,E1 89.771} C_DIS
LIN {X -0.077,Y -412.533,Z 1222.485,A 0.000,B 0.000,C 90.000,E1 87.364} C_DIS
LIN {X 0.068,Y -402.465,Z 1222.475,A 0.000,B 0.000,C 90.000,E1 85.412} C_DIS
LIN {X 0.007,Y -393.771,Z 1222.465,A 0.000,B 0.000,C 90.000,E1 83.742} C_DIS
LIN {X -0.172,Y -383.553,Z 1222.454,A 0.000,B 0.000,C 90.000,E1 81.781} C_DIS
LIN {X -0.081,Y -374.619,Z 1222.445,A 0.000,B 0.000,C 90.000,E1 80.038} C_DIS
LIN {X -0.085,Y -365.360,Z 1222.435,A 0.000,B 0.000,C 90.000,E1 78.285} C_DIS
LIN {X 0.173,Y -355.824,Z 1222.425,A 0.000,B 0.000,C 90.000,E1 76.464} C_DIS
LIN {X -0.079,Y -344.603,Z 1222.413,A 0.000,B 0.000,C 90.000,E1 74.393} C_DIS
LIN {X -0.164,Y -331.798,Z 1222.400,A 0.000,B 0.000,C 90.000,E1 71.945} C_DIS
LIN {X 0.055,Y -319.336,Z 1222.385,A 0.000,B 0.000,C 90.000,E1 69.390} C_DIS
LIN {X 0.027,Y -303.267,Z 1222.366,A 0.000,B 0.000,C 90.000,E1 65.845} C_DIS
LIN {X -0.148,Y -288.588,Z 1222.346,A 0.000,B 0.000,C 90.000,E1 62.231} C_DIS
LIN {X 0.043,Y -276.232,Z 1222.327,A 0.000,B 0.000,C 90.000,E1 58.791} C_DIS
LIN {X 0.052,Y -264.908,Z 1222.307,A 0.000,B 0.000,C 90.000,E1 55.308} C_DIS
LIN {X -0.033,Y -254.435,Z 1222.288,A 0.000,B 0.000,C 90.000,E1 51.778} C_DIS
LIN {X -0.043,Y -244.743,Z 1222.267,A 0.000,B 0.000,C 90.000,E1 48.162} C_DIS
LIN {X 0.015,Y -237.381,Z 1222.251,A 0.000,B 0.000,C 90.000,E1 45.202} C_DIS
LIN {X 0.048,Y -230.342,Z 1222.234,A 0.000,B 0.000,C 90.000,E1 42.204} C_DIS
LIN {X 0.000,Y -221.886,Z 1222.213,A 0.000,B 0.000,C 90.000,E1 38.418} C_DIS
LIN {X 0.080,Y -214.216,Z 1222.192,A 0.000,B 0.000,C 90.000,E1 34.532} C_DIS
LIN {X 0.133,Y -207.585,Z 1222.170,A 0.000,B 0.000,C 90.000,E1 30.590} C_DIS
LIN {X 0.105,Y -201.976,Z 1222.148,A 0.000,B 0.000,C 90.000,E1 26.616} C_DIS
LIN {X -0.085,Y -197.199,Z 1222.126,A 0.000,B 0.000,C 90.000,E1 22.642} C_DIS
LIN {X -0.059,Y -192.599,Z 1222.099,A 0.000,B 0.000,C 90.000,E1 17.747} C_DIS
LIN {X 0.075,Y -189.230,Z 1222.071,A 0.000,B 0.000,C 90.000,E1 12.771} C_DIS
LIN {X 0.062,Y -186.714,Z 1222.034,A 0.000,B 0.000,C 90.000,E1 6.144} C_DIS
LIN {X 0.062,Y -188.002,Z 1221.974,A 0.000,B 0.000,C 90.000,E1 355.355} C_DIS
LIN {X 0.005,Y -191.243,Z 1221.942,A 0.000,B 0.000,C 90.000,E1 349.577} C_DIS
LIN {X 0.069,Y -195.425,Z 1221.915,A 0.000,B 0.000,C 90.000,E1 344.629} C_DIS
LIN {X 0.099,Y -199.825,Z 1221.892,A 0.000,B 0.000,C 90.000,E1 340.550} C_DIS
LIN {X 0.037,Y -205.026,Z 1221.870,A 0.000,B 0.000,C 90.000,E1 336.538} C_DIS
LIN {X 0.003,Y -210.882,Z 1221.848,A 0.000,B 0.000,C 90.000,E1 332.564} C_DIS
LIN {X 0.020,Y -215.860,Z 1221.830,A 0.000,B 0.000,C 90.000,E1 329.410} C_DIS
LIN {X 0.037,Y -222.628,Z 1221.808,A 0.000,B 0.000,C 90.000,E1 325.515} C_DIS
LIN {X -0.030,Y -230.105,Z 1221.787,A 0.000,B 0.000,C 90.000,E1 321.698} C_DIS
LIN {X -0.011,Y -238.407,Z 1221.766,A 0.000,B 0.000,C 90.000,E1 317.919} C_DIS
LIN {X -0.082,Y -246.915,Z 1221.748,A 0.000,B 0.000,C 90.000,E1 314.595} C_DIS
LIN {X -0.072,Y -255.733,Z 1221.731,A 0.000,B 0.000,C 90.000,E1 311.676} C_DIS
LIN {X -0.151,Y -265.968,Z 1221.716,A 0.000,B 0.000,C 90.000,E1 308.830} C_DIS
LIN {X 0.117,Y -274.440,Z 1221.704,A 0.000,B 0.000,C 90.000,E1 306.664} C_DIS
LIN {X 0.083,Y -287.122,Z 1221.688,A 0.000,B 0.000,C 90.000,E1 303.913} C_DIS
LIN {X -0.108,Y -303.053,Z 1221.672,A 0.000,B 0.000,C 90.000,E1 300.924} C_DIS
LIN {X -0.004,Y -310.805,Z 1221.664,A 0.000,B 0.000,C 90.000,E1 299.589} C_DIS
LIN {X 0.118,Y -317.406,Z 1221.659,A 0.000,B 0.000,C 90.000,E1 298.615} C_DIS
LIN {X 0.030,Y -334.966,Z 1221.647,A 0.000,B 0.000,C 90.000,E1 296.411} C_DIS
LIN {X -0.064,Y -350.863,Z 1221.637,A 0.000,B 0.000,C 90.000,E1 294.591} C_DIS
LIN {X -0.080,Y -372.106,Z 1221.624,A 0.000,B 0.000,C 90.000,E1 292.280} C_DIS
LIN {X -0.050,Y -385.097,Z 1221.616,A 0.000,B 0.000,C 90.000,E1 290.918} C_DIS
LIN {X 0.080,Y -400.809,Z 1221.607,A 0.000,B 0.000,C 90.000,E1 289.268} C_DIS
LIN {X -0.218,Y -413.601,Z 1221.600,A 0.000,B 0.000,C 90.000,E1 288.000} C_DIS
LIN {X 0.048,Y -423.557,Z 1221.594,A 0.000,B 0.000,C 90.000,E1 286.913} C_DIS
LIN {X -0.168,Y -430.672,Z 1221.589,A 0.000,B 0.000,C 90.000,E1 286.134} C_DIS
LIN {X 0.050,Y -437.271,Z 1221.585,A 0.000,B 0.000,C 90.000,E1 285.300} C_DIS
LIN {X -0.200,Y -443.241,Z 1221.581,A 0.000,B 0.000,C 90.000,E1 284.537} C_DIS
LIN {X 0.030,Y -448.619,Z 1221.576,A 0.000,B 0.000,C 90.000,E1 283.716} C_DIS
LIN {X -0.013,Y -453.414,Z 1221.572,A 0.000,B 0.000,C 90.000,E1 282.939} C_DIS
LIN {X -0.129,Y -457.433,Z 1221.568,A 0.000,B 0.000,C 90.000,E1 282.175} C_DIS
LIN {X -0.127,Y -459.746,Z 1221.565,A 0.000,B 0.000,C 90.000,E1 281.658} C_DIS
LIN {X -0.016,Y -461.779,Z 1221.562,A 0.000,B 0.000,C 90.000,E1 281.130} C_DIS
LIN {X 0.101,Y -463.583,Z 1221.559,A 0.000,B 0.000,C 90.000,E1 280.602} C_DIS
LIN {X 0.145,Y -465.078,Z 1221.556,A 0.000,B 0.000,C 90.000,E1 280.084} C_DIS
LIN {X -0.176,Y -466.306,Z 1221.553,A 0.000,B 0.000,C 90.000,E1 279.613} C_DIS
LIN {X -0.108,Y -467.269,Z 1221.550,A 0.000,B 0.000,C 90.000,E1 279.095} C_DIS
LIN {X 0.041,Y -467.946,Z 1221.548,A 0.000,B 0.000,C 90.000,E1 278.568} C_DIS
LIN {X 0.125,Y -468.351,Z 1221.545,A 0.000,B 0.000,C 90.000,E1 278.049} C_DIS
LIN {X -0.249,Y -468.446,Z 1221.542,A 0.000,B 0.000,C 90.000,E1 277.587} C_DIS
LIN {X -0.156,Y -468.160,Z 1221.539,A 0.000,B 0.000,C 90.000,E1 277.068} C_DIS
LIN {X -0.061,Y -467.465,Z 1221.536,A 0.000,B 0.000,C 90.000,E1 276.549} C_DIS
LIN {X 0.033,Y -466.421,Z 1221.534,A 0.000,B 0.000,C 90.000,E1 276.030} C_DIS
LIN {X 0.121,Y -464.902,Z 1221.531,A 0.000,B 0.000,C 90.000,E1 275.511} C_DIS
LIN {X 0.025,Y -461.853,Z 1221.526,A 0.000,B 0.000,C 90.000,E1 274.759} C_DIS
LIN {X 0.049,Y -459.109,Z 1221.524,A 0.000,B 0.000,C 90.000,E1 274.245} C_DIS
LIN {X -0.138,Y -457.512,Z 1221.522,A 0.000,B 0.000,C 90.000,E1 274.012} C_DIS
LIN {X -0.133,Y -453.617,Z 1221.519,A 0.000,B 0.000,C 90.000,E1 273.498} C_DIS
LIN {X -0.120,Y -448.711,Z 1221.516,A 0.000,B 0.000,C 90.000,E1 272.980} C_DIS
LIN {X 0.147,Y -445.859,Z 1221.515,A 0.000,B 0.000,C 90.000,E1 272.694} C_DIS
LIN {X -0.031,Y -442.662,Z 1221.514,A 0.000,B 0.000,C 90.000,E1 272.465} C_DIS
LIN {X 0.182,Y -436.020,Z 1221.511,A 0.000,B 0.000,C 90.000,E1 272.007} C_DIS
LIN {X 0.079,Y -428.882,Z 1221.509,A 0.000,B 0.000,C 90.000,E1 271.661} C_DIS
LIN {X 0.057,Y -421.621,Z 1221.508,A 0.000,B 0.000,C 90.000,E1 271.375} C_DIS
LIN {X 0.105,Y -411.514,Z 1221.506,A 0.000,B 0.000,C 90.000,E1 271.031} C_DIS
LIN {X 0.115,Y -400.835,Z 1221.504,A 0.000,B 0.000,C 90.000,E1 270.745} C_DIS
LIN {X -0.187,Y -393.877,Z 1221.503,A 0.000,B 0.000,C 90.000,E1 270.630} C_DIS
LIN {X 0.034,Y -385.320,Z 1221.503,A 0.000,B 0.000,C 90.000,E1 270.458} C_DIS
LIN {X 0.092,Y -375.323,Z 1221.502,A 0.000,B 0.000,C 90.000,E1 270.344} C_DIS
LIN {X 0.140,Y -366.882,Z 1221.502,A 0.000,B 0.000,C 90.000,E1 270.286} C_DIS
LIN {X 0.075,Y -362.190,Z 1221.502,A 0.000,B 0.000,C 90.000,E1 270.286} C_DIS
LIN {X 0.006,Y -181.581,Z 1221.502,A 0.000,B 0.000,C 90.000,E1 270.286} C_DIS
LIN {X -0.013,Y -180.833,Z 1221.472,A 0.000,B 0.000,C 90.000,E1 264.894} C_DIS
LIN {X 0.066,Y -178.940,Z 1221.443,A 0.000,B 0.000,C 90.000,E1 259.803} C_DIS
LIN {X -0.066,Y -175.989,Z 1221.415,A 0.000,B 0.000,C 90.000,E1 254.755} C_DIS
LIN {X 0.048,Y -175.489,Z 1221.410,A 0.000,B 0.000,C 90.000,E1 253.866} C_DIS
LIN {X -0.057,Y -172.234,Z 1221.387,A 0.000,B 0.000,C 90.000,E1 249.625} C_DIS
LIN {X -0.079,Y -171.711,Z 1221.382,A 0.000,B 0.000,C 90.000,E1 248.773} C_DIS
LIN {X 0.006,Y -167.306,Z 1221.353,A 0.000,B 0.000,C 90.000,E1 243.563} C_DIS
LIN {X 0.013,Y -166.685,Z 1221.348,A 0.000,B 0.000,C 90.000,E1 242.692} C_DIS
LIN {X 0.003,Y -162.668,Z 1221.324,A 0.000,B 0.000,C 90.000,E1 238.329} C_DIS
LIN {X -0.024,Y -161.358,Z 1221.314,A 0.000,B 0.000,C 90.000,E1 236.580} C_DIS
LIN {X 0.011,Y -157.351,Z 1221.290,A 0.000,B 0.000,C 90.000,E1 232.145} C_DIS
LIN {X 0.039,Y -155.339,Z 1221.275,A 0.000,B 0.000,C 90.000,E1 229.461} C_DIS
LIN {X -0.030,Y -151.686,Z 1221.250,A 0.000,B 0.000,C 90.000,E1 225.000} C_DIS
LIN {X 0.017,Y -150.550,Z 1221.240,A 0.000,B 0.000,C 90.000,E1 223.176} C_DIS
LIN {X 0.050,Y -147.277,Z 1221.215,A 0.000,B 0.000,C 90.000,E1 218.624} C_DIS
LIN {X 0.022,Y -145.305,Z 1221.194,A 0.000,B 0.000,C 90.000,E1 214.978} C_DIS
LIN {X 0.014,Y -142.397,Z 1221.164,A 0.000,B 0.000,C 90.000,E1 209.461} C_DIS
LIN {X -0.003,Y -141.378,Z 1221.148,A 0.000,B 0.000,C 90.000,E1 206.693} C_DIS
LIN {X 0.038,Y -139.348,Z 1221.112,A 0.000,B 0.000,C 90.000,E1 200.174} C_DIS
LIN {X -0.020,Y -138.784,Z 1221.097,A 0.000,B 0.000,C 90.000,E1 197.402} C_DIS
LIN {X 0.039,Y -138.344,Z 1221.055,A 0.000,B 0.000,C 90.000,E1 189.905} C_DIS
LIN {X 0.059,Y -139.389,Z 1221.008,A 0.000,B 0.000,C 90.000,E1 181.489} C_DIS
LIN {X -0.028,Y -141.286,Z 1220.972,A 0.000,B 0.000,C 90.000,E1 175.008} C_DIS
LIN {X -0.070,Y -142.650,Z 1220.957,A 0.000,B 0.000,C 90.000,E1 172.243} C_DIS
LIN {X 0.022,Y -144.986,Z 1220.931,A 0.000,B 0.000,C 90.000,E1 167.589} C_DIS
LIN {X 0.012,Y -147.614,Z 1220.911,A 0.000,B 0.000,C 90.000,E1 163.921} C_DIS
LIN {X -0.051,Y -150.238,Z 1220.890,A 0.000,B 0.000,C 90.000,E1 160.296} C_DIS
LIN {X -0.036,Y -153.632,Z 1220.870,A 0.000,B 0.000,C 90.000,E1 156.666} C_DIS
LIN {X 0.023,Y -157.046,Z 1220.850,A 0.000,B 0.000,C 90.000,E1 153.050} C_DIS
LIN {X 0.021,Y -161.173,Z 1220.831,A 0.000,B 0.000,C 90.000,E1 149.488} C_DIS
LIN {X -0.036,Y -163.269,Z 1220.821,A 0.000,B 0.000,C 90.000,E1 147.740} C_DIS
LIN {X 0.062,Y -167.709,Z 1220.801,A 0.000,B 0.000,C 90.000,E1 144.196} C_DIS
LIN {X -0.025,Y -171.529,Z 1220.787,A 0.000,B 0.000,C 90.000,E1 141.618} C_DIS
LIN {X 0.018,Y -176.469,Z 1220.768,A 0.000,B 0.000,C 90.000,E1 138.162} C_DIS
LIN {X 0.017,Y -180.765,Z 1220.753,A 0.000,B 0.000,C 90.000,E1 135.607} C_DIS
LIN {X 0.006,Y -186.171,Z 1220.735,A 0.000,B 0.000,C 90.000,E1 132.243} C_DIS
LIN {X 0.070,Y -190.808,Z 1220.721,A 0.000,B 0.000,C 90.000,E1 129.725} C_DIS
LIN {X -0.011,Y -196.566,Z 1220.703,A 0.000,B 0.000,C 90.000,E1 126.457} C_DIS
LIN {X 0.083,Y -201.116,Z 1220.690,A 0.000,B 0.000,C 90.000,E1 124.119} C_DIS
LIN {X 0.094,Y -310.296,Z 1220.690,A 0.000,B 0.000,C 90.000,E1 124.119} C_DIS
LIN {X 0.115,Y -315.409,Z 1220.689,A 0.000,B 0.000,C 90.000,E1 123.992} C_DIS
LIN {X -0.047,Y -317.975,Z 1220.688,A 0.000,B 0.000,C 90.000,E1 123.865} C_DIS
LIN {X -0.075,Y -321.755,Z 1220.686,A 0.000,B 0.000,C 90.000,E1 123.499} C_DIS
LIN {X -0.129,Y -325.235,Z 1220.683,A 0.000,B 0.000,C 90.000,E1 122.959} C_DIS
LIN {X -0.041,Y -326.645,Z 1220.681,A 0.000,B 0.000,C 90.000,E1 122.625} C_DIS
LIN {X 0.105,Y -338.669,Z 1220.664,A 0.000,B 0.000,C 90.000,E1 119.461} C_DIS
LIN {X 0.104,Y -350.917,Z 1220.648,A 0.000,B 0.000,C 90.000,E1 116.693} C_DIS
LIN {X -0.020,Y -364.646,Z 1220.633,A 0.000,B 0.000,C 90.000,E1 114.003} C_DIS
LIN {X 0.003,Y -378.194,Z 1220.620,A 0.000,B 0.000,C 90.000,E1 111.642} C_DIS
LIN {X 0.093,Y -393.105,Z 1220.607,A 0.000,B 0.000,C 90.000,E1 109.322} C_DIS
LIN {X -0.075,Y -409.483,Z 1220.595,A 0.000,B 0.000,C 90.000,E1 107.094} C_DIS
LIN {X -0.074,Y -427.445,Z 1220.583,A 0.000,B 0.000,C 90.000,E1 104.898} C_DIS
LIN {X -0.039,Y -446.972,Z 1220.571,A 0.000,B 0.000,C 90.000,E1 102.771} C_DIS
LIN {X 0.183,Y -467.233,Z 1220.560,A 0.000,B 0.000,C 90.000,E1 100.782} C_DIS
LIN {X 0.240,Y -472.339,Z 1220.557,A 0.000,B 0.000,C 90.000,E1 100.310} C_DIS
LIN {X -0.263,Y -474.354,Z 1220.556,A 0.000,B 0.000,C 90.000,E1 100.141} C_DIS
LIN {X 0.067,Y -476.020,Z 1220.555,A 0.000,B 0.000,C 90.000,E1 99.849} C_DIS
LIN {X -0.073,Y -477.272,Z 1220.553,A 0.000,B 0.000,C 90.000,E1 99.613} C_DIS
LIN {X 0.061,Y -478.810,Z 1220.551,A 0.000,B 0.000,C 90.000,E1 99.095} C_DIS
LIN {X -0.196,Y -479.299,Z 1220.548,A 0.000,B 0.000,C 90.000,E1 98.624} C_DIS
LIN {X -0.044,Y -478.816,Z 1220.545,A 0.000,B 0.000,C 90.000,E1 98.106} C_DIS
LIN {X 0.113,Y -477.291,Z 1220.542,A 0.000,B 0.000,C 90.000,E1 97.587} C_DIS
LIN {X -0.016,Y -476.057,Z 1220.541,A 0.000,B 0.000,C 90.000,E1 97.352} C_DIS
LIN {X 0.128,Y -472.510,Z 1220.538,A 0.000,B 0.000,C 90.000,E1 96.834} C_DIS
LIN {X -0.186,Y -456.157,Z 1220.525,A 0.000,B 0.000,C 90.000,E1 94.588} C_DIS
LIN {X 0.112,Y -438.848,Z 1220.511,A 0.000,B 0.000,C 90.000,E1 91.949} C_DIS
LIN {X 0.068,Y -425.968,Z 1220.499,A 0.000,B 0.000,C 90.000,E1 89.828} C_DIS
LIN {X -0.169,Y -412.628,Z 1220.486,A 0.000,B 0.000,C 90.000,E1 87.421} C_DIS
LIN {X 0.062,Y -401.107,Z 1220.473,A 0.000,B 0.000,C 90.000,E1 85.179} C_DIS
LIN {X 0.000,Y -390.943,Z 1220.462,A 0.000,B 0.000,C 90.000,E1 83.223} C_DIS
LIN {X 0.195,Y -380.690,Z 1220.451,A 0.000,B 0.000,C 90.000,E1 81.197} C_DIS
LIN {X -0.135,Y -371.665,Z 1220.442,A 0.000,B 0.000,C 90.000,E1 79.511} C_DIS
LIN {X 0.166,Y -362.303,Z 1220.432,A 0.000,B 0.000,C 90.000,E1 77.701} C_DIS
LIN {X -0.040,Y -351.125,Z 1220.420,A 0.000,B 0.000,C 90.000,E1 75.644} C_DIS
LIN {X 0.027,Y -339.875,Z 1220.408,A 0.000,B 0.000,C 90.000,E1 73.504} C_DIS
LIN {X -0.079,Y -327.206,Z 1220.395,A 0.000,B 0.000,C 90.000,E1 71.040} C_DIS
LIN {X -0.005,Y -311.945,Z 1220.377,A 0.000,B 0.000,C 90.000,E1 67.847} C_DIS
LIN {X -0.029,Y -297.848,Z 1220.359,A 0.000,B 0.000,C 90.000,E1 64.588} C_DIS
LIN {X -0.098,Y -284.850,Z 1220.340,A 0.000,B 0.000,C 90.000,E1 61.257} C_DIS
LIN {X 0.113,Y -272.740,Z 1220.321,A 0.000,B 0.000,C 90.000,E1 57.788} C_DIS
LIN {X -0.116,Y -262.723,Z 1220.304,A 0.000,B 0.000,C 90.000,E1 54.689} C_DIS
LIN {X 0.053,Y -252.364,Z 1220.284,A 0.000,B 0.000,C 90.000,E1 51.090} C_DIS
LIN {X -0.019,Y -242.768,Z 1220.264,A 0.000,B 0.000,C 90.000,E1 47.472} C_DIS
LIN {X -0.085,Y -233.653,Z 1220.243,A 0.000,B 0.000,C 90.000,E1 43.785} C_DIS
LIN {X 0.029,Y -226.679,Z 1220.226,A 0.000,B 0.000,C 90.000,E1 40.744} C_DIS
LIN {X -0.097,Y -218.460,Z 1220.205,A 0.000,B 0.000,C 90.000,E1 36.950} C_DIS
LIN {X -0.064,Y -212.570,Z 1220.188,A 0.000,B 0.000,C 90.000,E1 33.833} C_DIS
LIN {X 0.011,Y -206.146,Z 1220.166,A 0.000,B 0.000,C 90.000,E1 29.873} C_DIS
LIN {X -0.058,Y -200.732,Z 1220.144,A 0.000,B 0.000,C 90.000,E1 25.899} C_DIS
LIN {X -0.004,Y -196.126,Z 1220.121,A 0.000,B 0.000,C 90.000,E1 21.844} C_DIS
LIN {X -0.002,Y -192.333,Z 1220.099,A 0.000,B 0.000,C 90.000,E1 17.764} C_DIS
LIN {X -0.006,Y -188.941,Z 1220.071,A 0.000,B 0.000,C 90.000,E1 12.827} C_DIS
LIN {X -0.036,Y -186.405,Z 1220.034,A 0.000,B 0.000,C 90.000,E1 6.201} C_DIS
LIN {X 0.051,Y -187.670,Z 1219.974,A 0.000,B 0.000,C 90.000,E1 355.355} C_DIS
LIN {X 0.015,Y -190.925,Z 1219.942,A 0.000,B 0.000,C 90.000,E1 349.567} C_DIS
LIN {X 0.032,Y -195.127,Z 1219.915,A 0.000,B 0.000,C 90.000,E1 344.629} C_DIS
LIN {X 0.052,Y -199.563,Z 1219.892,A 0.000,B 0.000,C 90.000,E1 340.550} C_DIS
LIN {X -0.019,Y -204.776,Z 1219.870,A 0.000,B 0.000,C 90.000,E1 336.538} C_DIS
LIN {X 0.035,Y -210.654,Z 1219.848,A 0.000,B 0.000,C 90.000,E1 332.538} C_DIS
LIN {X -0.053,Y -215.643,Z 1219.830,A 0.000,B 0.000,C 90.000,E1 329.410} C_DIS
LIN {X -0.046,Y -222.419,Z 1219.808,A 0.000,B 0.000,C 90.000,E1 325.515} C_DIS
LIN {X 0.021,Y -229.912,Z 1219.787,A 0.000,B 0.000,C 90.000,E1 321.662} C_DIS
LIN {X 0.066,Y -238.233,Z 1219.766,A 0.000,B 0.000,C 90.000,E1 317.877} C_DIS
LIN {X -0.018,Y -246.788,Z 1219.748,A 0.000,B 0.000,C 90.000,E1 314.555} C_DIS
LIN {X 0.003,Y -255.656,Z 1219.731,A 0.000,B 0.000,C 90.000,E1 311.634} C_DIS
LIN {X 0.160,Y -267.316,Z 1219.713,A 0.000,B 0.000,C 90.000,E1 308.382} C_DIS
LIN {X 0.076,Y -275.961,Z 1219.702,A 0.000,B 0.000,C 90.000,E1 306.297} C_DIS
LIN {X -0.085,Y -288.822,Z 1219.686,A 0.000,B 0.000,C 90.000,E1 303.579} C_DIS
LIN {X 0.035,Y -304.906,Z 1219.670,A 0.000,B 0.000,C 90.000,E1 300.541} C_DIS
LIN {X 0.124,Y -310.768,Z 1219.664,A 0.000,B 0.000,C 90.000,E1 299.539} C_DIS
LIN {X -0.071,Y -317.439,Z 1219.659,A 0.000,B 0.000,C 90.000,E1 298.615} C_DIS
LIN {X 0.150,Y -334.946,Z 1219.647,A 0.000,B 0.000,C 90.000,E1 296.360} C_DIS
LIN {X 0.049,Y -353.407,Z 1219.635,A 0.000,B 0.000,C 90.000,E1 294.259} C_DIS
LIN {X 0.074,Y -374.637,Z 1219.622,A 0.000,B 0.000,C 90.000,E1 291.972} C_DIS
LIN {X 0.030,Y -387.785,Z 1219.615,A 0.000,B 0.000,C 90.000,E1 290.610} C_DIS
LIN {X 0.222,Y -403.530,Z 1219.605,A 0.000,B 0.000,C 90.000,E1 288.960} C_DIS
LIN {X -0.018,Y -413.795,Z 1219.600,A 0.000,B 0.000,C 90.000,E1 287.946} C_DIS
